lreal1:=fbMeter[1].stDataEMOutPowerDelay.lrPowerTotal;
lreal2:=fbMeter[2].stDataEMOutPowerDelay.lrPowerTotal;
lreal3:=fbMeter[3].stDataEMOutPowerDelay.lrPowerTotal;
lreal4:=fbMeter[4].stDataEMOutPowerDelay.lrPowerTotal;
lreal5:=fbMeter[5].stDataEMOutPowerDelay.lrPowerTotal;
lreal6:=fbMeter[6].stDataEMOutPowerDelay.lrPowerTotal;
lreal7:=fbMeter[7].stDataEMOutPowerDelay.lrPowerTotal;
lreal8:=fbMeter[8].stDataEMOutPowerDelay.lrPowerTotal;
lreal9:=fbMeter[9].stDataEMOutPowerDelay.lrPowerTotal;
lreal10:=fbMeter[10].stDataEMOutPowerDelay.lrPowerTotal;
lreal11:=fbMeter[11].stDataEMOutPowerDelay.lrPowerTotal;
lreal12:=fbMeter[12].stDataEMOutPowerDelay.lrPowerTotal;
lreal13:=fbMeter[13].stDataEMOutPowerDelay.lrPowerTotal;
lreal14:=fbMeter[14].stDataEMOutPowerDelay.lrPowerTotal;
lreal15:=fbMeter[15].stDataEMOutPowerDelay.lrPowerTotal;
lreal16:=fbMeter[16].stDataEMOutPowerDelay.lrPowerTotal;
lreal17:=fbMeter[17].stDataEMOutPowerDelay.lrPowerTotal;
lreal18:=fbMeter[18].stDataEMOutPowerDelay.lrPowerTotal;
lreal19:=fbMeter[19].stDataEMOutPowerDelay.lrPowerTotal;
lreal20:=fbMeter[20].stDataEMOutPowerDelay.lrPowerTotal;

(*----------------------------------------------------------Save persistent data----------------------------------------------------------------*)

// arrPD[1](lrValue:= BOOL_TO_LREAL(bEnable), bEventBasedActive=> );
// arrPD[2](lrValue:= BYTE_TO_LREAL(byAmountOfInverters), bEventBasedActive=> );
PD_String(sText:= sIPAdress, bEventBasedActive=> );

END_FUNCTION_BLOCK

// ---- FBs/Keba/FB_ECS_Keba_P30.TcPOU
FUNCTION_BLOCK FB_ECS_Keba_P30
VAR_INPUT PERSISTENT
	///{#lynus.ag#()} //Enable the Fuctionblock and his logic
	bEnable: BOOL;
	///With True its possible to invert all received power data from the electric meter
	bPowerDataInvers: BOOL;
	///Electric Fuse Line on wich the ECS is connected => 1 2 3 (If 0 then this charging station is not connected to a Electric Fuse Line)
	byElectricFuseLine: BYTE;
	///Failsafe Current when the connection between PLC and Charging station is interrupted. 0mA = CS Off, 6000mA - 32000mA
	uiFailsafeCurrent: UINT;
	///Failsafe Timeout when the connection between PLC and Charging station is interrupted. 10 - 600 sec
	uiFailsafeTimeOut: UINT := 10;
	///Number of EMS what control this Device.
	diNrOfEMS_IN: DINT;
	///Number of the electric meter for incoming power data. (Power Data for this Device)
	diNrOfEM_IN_CS: DINT;
	///IP Adress from the Keba charging station
	sIPAdress: STRING(15);
	///{#lynus.ag#()} //Setup charging station
	stSetupECS: ST_Setup_ECS;
END_VAR
VAR_OUTPUT
	///{#lynus.ag#()} //Electric charging station output data
	stDataECS: ST_ECS_Output;
	///Active Number from the Electric charging Function for using on other functions
	diNrOfECS_OUT: DINT;
	///Total Electric Power in kW read out directly from the Charging station. (Real time)
	lrTotalPowerECSRealTime: LREAL;
END_VAR
VAR
	///Function block for electric charging station
	{attribute 'hide' := ''}
	fbCS: FB_ElectricChargingStation;
	///Function block to calcualte the number of the Device
	{attribute 'hide' := ''}
	fbNumberDevice: FB_NumberOfDevice;
	///Digital Input from external loock signal
	fbDIExternalLock: FB_XL1XXX_DI;
	///Modbus Read Function (FC3)
	{attribute 'hide' := ''}
	fbMBRead_FC3: FB_MBReadRegs;
	///Modbus Write Function (FC6)
	{attribute 'hide' := ''}
	fbMBWrite_FC6: FB_MBWriteSingleReg;
	///Convert Word to Dword
	{attribute 'hide' := ''}
	fbConvertWordToDword: FB_CV_WORD_TO_DWORD;
	///Timer for Delay between Requests
	{attribute 'hide' := ''}
	timDelay: TON;
	///Timer for Timeout
	{attribute 'hide' := ''}
	timTimeout: TON;
	///Timer to dissable the Function after Lynus_Standards.Constants_General.tTimeDissableLynusFunctions Days without connection to the Lynus Cloud
	{attribute 'hide' := ''}
	timDissableFunctions: TON;
	///Timer to try reset the connection Flag on the GVL. (When somebody delete the Connection Function and make only a onlinechange)
	{attribute 'hide' := ''}
	timResetConnectionOnGVL: TON;
	///Charging Time
	{attribute 'hide' := ''}
	timChTimeSocket: TON;
	///Timer to start the state machine with Daley after enabling or after the system ist restartet
	{attribute 'hide' := ''}
	timDelayStart: TON;
	///Timer to Close the Socket after to much Errors
	{attribute 'hide' := ''}
	timCloseSocket: TON;
	///Internal positive Edge
	{attribute 'hide' := ''}
	FPError_FC_3: R_TRIG;
	///Internal positive Edge
	{attribute 'hide' := ''}
	FPError_FC_6: R_TRIG;
	///Internal positive Edge
	{attribute 'hide' := ''}
	FPEnable: R_TRIG;
	///Function to save persistent data
	{attribute 'hide' := ''}
	arrPD: ARRAY[1..16] OF FB_PersistentData_Number;
	///Function to save persistent string data
	{attribute 'hide' := ''}
	fbPDString: FB_PersistentData_String;
	///Buffer with Data from FC3
	{attribute 'hide' := ''}
	arrBuffer_FC3: ARRAY[1..2] OF WORD;
	///Error State from the charging station
	{attribute 'hide' := ''}
	bErrorCS: BOOL;
	///Modbus TCP Function Error Counter																	
	{attribute 'hide' := ''}
	byMBTCPErrorCounter: BYTE;
	///Wait in Step before start to clean data on PLC
	{attribute 'hide' := ''}
	byWaitInStep: BYTE;
	///State machine to handle the data on the GVL
	{attribute 'hide' := ''}
	iStateGVLData: INT;
	///State machine for read out Data over Modbus TCP
	{attribute 'hide' := ''}
	iStateModbusRead: INT;
	///State machine for write Data over Modbus TCP
	{attribute 'hide' := ''}
	iStateModbusWrite: INT;
	///State machine for error out Data over Modbus TCP	
	{attribute 'hide' := ''}
	iStateModbusError: INT;
	///Variable to compare the state machine variable to set or reset the timeout timer
	{attribute 'hide' := ''}
	iStateModbus_CP: INT;
	///Number of active batterys
	{attribute 'hide' := ''}
	diNumberOfActiveBatterys: DINT;
	///Number of battery inverters that work in Emergency Power operation 
	{attribute 'hide' := ''}
	diNumberOfBatteryInverterInEPO: DINT;
	///Loop to clean old data on GVL
	{attribute 'hide' := ''}
	diLPForGVL: DINT;
	///Counter to clean old data on GVL
	{attribute 'hide' := ''}
	diCounterForGVL: DINT;
	///Sum of the SOC from all batterys
	{attribute 'hide' := ''}
	dwSumSOC: DWORD;
	///Charging State from the Keba Charger
	{attribute 'hide' := ''}
	dwChargingState: DWORD;
	///Cable State from the Keba Charger
	{attribute 'hide' := ''}
	dwCableState: DWORD;
	///Error Code from the Keba Charger
	{attribute 'hide' := ''}
	dwErrorCode: DWORD;
	///Power from the ECS in W 
	{attribute 'hide' := ''}
	rPowerECS: REAL;
	///Energy Counter Consumption in Wh
	{attribute 'hide' := ''}
	lrTotalCounterEnergy_Consumption: LREAL;
	///Charged Energy from the active Session in Wh
	{attribute 'hide' := ''}
	lrChargedEnergySession: LREAL;
	///Loop to check some data from batterys
	{attribute 'hide' := ''}
	liLPBatteryData: LINT;
	///Loop to check if 1 or more battery inverters build a island grid
	{attribute 'hide' := ''}
	liLPInEPO: LINT;
END_VAR
VAR PERSISTENT
	///Number of EMS what control this Device to compare with the original
	{attribute 'conditionalshow' := ''}
	diNrOfEMS_IN_CP: DINT;
END_VAR

//Creator : Kai Ebensperger
//Company : Lynus AG
//Date : 15.07.2022
//Version : 1.0.0.0

//With this Funcition its possible to communicate with a Keba P30 Charging station over Modbus TCP.
//Support the C-Series from Version 3.10.16 or higher
//Support the X-Series from Version 1.11 or higher
//Its possible to controll the charging station over the charge current
//When the Function send 0 Ampere is switched of, then the charging station is blocked and its not possible to charge
//The Communication is not so fast because in the Documentation they write that we can read every 500MS but we can write onle ever 5 seconds.
//We can read only 1 Register at each command. Its not possible to read more Registers with 1 command
//The Unit ID is always 255
//Also the Settings for Fail Save is includes in ths Fuction. The Failsave Current is set to uiFailsafeCurrent.
//Failsafe takes effect when the connection between the PLC and the charging station is interrupted. Timout is uiFailsafeTimeOut in seconds.

//Versions that are supported : 1.3

//NOTE for diNr.....Designation => 
//_IN = Here Data come in from other Functions or go out to other functions about the GVL
//_OUT = Here Data go out to other functions about the GVL

(*--------------------------------------------------------------------------------------------Limits-------------------------------------------------------------------------------------*)

diNrOfEMS_IN := LIMIT(0,diNrOfEMS_IN,Constants_Energy.diMaxNumberOfEMS);
	diNrOfEM_IN_CS := LIMIT(0,diNrOfEM_IN_CS,Constants_Energy.diMaxNumberOfElectricMeters);
		byElectricFuseLine := LIMIT(0,byElectricFuseLine,30);
			IF uiFailsafeCurrent > 0 THEN 
				uiFailsafeCurrent := LIMIT(6000,uiFailsafeCurrent,32000);
			END_IF 
				uiFailsafeTimeOut := LIMIT(10,uiFailsafeTimeOut,600);	
		
(*------------------------------------------------------------------Power Data----------------------------------------------------------------------------*)

IF diNrOfEM_IN_CS <> 0 THEN
	//Energy Session Input data
	fbCS.bCalculateEnergySession := FALSE;
	fbCS.arrSocketPowerECS[1] := 0;
	fbCS.arrSocketPowerECS[2] := 0;
	fbCS.arrSocketPowerECS[3] := 0;
	fbCS.arrSocketPowerECS[4] := 0;
	fbCS.arrSocketEnergySession[1] := 0;
	fbCS.arrSocketEnergySession[2] := 0;
	fbCS.arrSocketEnergySession[3] := 0;
	fbCS.arrSocketEnergySession[4] := 0;
		IF NOT bPowerDataInvers THEN
			//Energy meter input data for cs Function block
			fbCS.lrCounterEnergyT1_Consumption := Lynus_Standards.GVL_Energy.stDataElectricMeters[diNrOfEM_IN_CS].lrCounterEnergyT1_Production * 1000;
			fbCS.lrCounterEnergyT2_Consumption := Lynus_Standards.GVL_Energy.stDataElectricMeters[diNrOfEM_IN_CS].lrCounterEnergyT2_Production * 1000;
			fbCS.lrCounterEnergyT1_Production := Lynus_Standards.GVL_Energy.stDataElectricMeters[diNrOfEM_IN_CS].lrCounterEnergyT1_Consumption * 1000;
			fbCS.lrCounterEnergyT2_Production := Lynus_Standards.GVL_Energy.stDataElectricMeters[diNrOfEM_IN_CS].lrCounterEnergyT1_Consumption * 1000;
			fbCS.lrTotalCounterEnergy_Consumption := Lynus_Standards.GVL_Energy.stDataElectricMeters[diNrOfEM_IN_CS].lrTotalCounterEnergy_Production * 1000;
			fbCS.lrTotalCounterEnergy_Production := Lynus_Standards.GVL_Energy.stDataElectricMeters[diNrOfEM_IN_CS].lrTotalCounterEnergy_Consumption * 1000;
				fbCS.lrTotalPowerECS := (Lynus_Standards.GVL_Energy.stDataElectricMeters[diNrOfEM_IN_CS].lrPower * 1000) * - 1;
			ELSE
			//Energy meter input data for cs Function block
			fbCS.lrCounterEnergyT1_Consumption := Lynus_Standards.GVL_Energy.stDataElectricMeters[diNrOfEM_IN_CS].lrCounterEnergyT1_Consumption * 1000;
			fbCS.lrCounterEnergyT2_Consumption := Lynus_Standards.GVL_Energy.stDataElectricMeters[diNrOfEM_IN_CS].lrCounterEnergyT2_Consumption * 1000;
			fbCS.lrCounterEnergyT1_Production := Lynus_Standards.GVL_Energy.stDataElectricMeters[diNrOfEM_IN_CS].lrCounterEnergyT1_Production * 1000;
			fbCS.lrCounterEnergyT2_Production := Lynus_Standards.GVL_Energy.stDataElectricMeters[diNrOfEM_IN_CS].lrCounterEnergyT2_Production * 1000;
			fbCS.lrTotalCounterEnergy_Consumption := Lynus_Standards.GVL_Energy.stDataElectricMeters[diNrOfEM_IN_CS].lrTotalCounterEnergy_Consumption * 1000;
			fbCS.lrTotalCounterEnergy_Production := Lynus_Standards.GVL_Energy.stDataElectricMeters[diNrOfEM_IN_CS].lrTotalCounterEnergy_Production * 1000;
				fbCS.lrTotalPowerECS := Lynus_Standards.GVL_Energy.stDataElectricMeters[diNrOfEM_IN_CS].lrPower * 1000;
		END_IF
ELSE
	//Energy meter input data for cs Function block
	fbCS.lrCounterEnergyT1_Consumption := lrTotalCounterEnergy_Consumption;
	fbCS.lrCounterEnergyT2_Consumption := 0;
	fbCS.lrCounterEnergyT1_Production := 0;
	fbCS.lrCounterEnergyT2_Production := 0;
	fbCS.lrTotalCounterEnergy_Consumption := lrTotalCounterEnergy_Consumption;
	fbCS.lrTotalCounterEnergy_Production := 0;
		fbCS.lrTotalPowerECS := rPowerECS;
	//Energy Session Input data
	fbCS.bCalculateEnergySession := FALSE;
	fbCS.arrSocketPowerECS[1] := rPowerECS;
	fbCS.arrSocketPowerECS[2] := 0;
	fbCS.arrSocketPowerECS[3] := 0;
	fbCS.arrSocketPowerECS[4] := 0;
	fbCS.arrSocketEnergySession[1] := lrChargedEnergySession;
	fbCS.arrSocketEnergySession[2] := 0;
	fbCS.arrSocketEnergySession[3] := 0;
	fbCS.arrSocketEnergySession[4] := 0;
END_IF			

(*-------------------------------------------------------------Calcualte the number of ECS---------------------------------------------------------------*)

fbNumberDevice(
	diActualNumberOfDevices:= Lynus_Standards.GVL_Energy.stNumberOfDevices.diNumberOfECS, 
	diMaxNumberOfDevices:= Constants_Energy.diMaxNumberOfElectricChargingStations, 
	udiCounterOnlineChange:= TwinCAT_SystemInfoVarList._AppInfo.OnlineChangeCnt, 
	bNumberIsCalculatet=> , 
	bFPNumberIsCalculatet=> , 
	bOnlineChange=> , 
	diNumberForThisDevice=> diNrOfECS_OUT, 
	diNumberOfTotalDevices=> );

//Write new Numer on GVL
IF fbNumberDevice.bFPNumberIsCalculatet THEN
	Lynus_Standards.GVL_Energy.stNumberOfDevices.diNumberOfECS := fbNumberDevice.diNumberOfTotalDevices;	
END_IF 

//Delete old Number on GVL
IF fbNumberDevice.bOnlineChange THEN 
	Lynus_Standards.GVL_Energy.stNumberOfDevices.diNumberOfECS := diNrOfECS_OUT;	
		iStateGVLData := 1;
END_IF

(*-------------------------------------------------------------Service from Backend is ready and check the connection to backen for dissabel/enable Function---------------------------------------------------------------*)

//Try to reset the variable for connection on the GVL. When all is normal then the Lynus Mqtt connection function set this variable to true in the next cycle
//When we have no connection to the backend then after Lynus_Standards.Constants_General.tTimeDissableLynusFunctions days the Function is dissabled with all of his functionalities
timResetConnectionOnGVL(IN:= NOT timResetConnectionOnGVL.Q, PT:= T#1H, Q=> , ET=> );
	IF timResetConnectionOnGVL.Q THEN Lynus_Standards.GVL_Communicator.bStateConnectionToEnableFunctions := FALSE; END_IF
		IF NOT Lynus_Standards.GVL_Communicator.bStateConnectionToEnableFunctions THEN timDissableFunctions.IN := TRUE; ELSE timDissableFunctions.IN := FALSE; END_IF  
			timDissableFunctions(IN:= , PT:= Lynus_Standards.Constants_General.tTimeDissableLynusFunctions, Q=> , ET=> );
			
(*--------------------------------------------------------------------------------------------State Machine Read--------------------------------------------------------------------------------------*)

//Timer for Delay
timDelay(IN:= , PT:= T#750MS, Q=> , ET=> );

//Timer for Timeout in Statemachine
IF (iStateModbusRead > 0 AND iStateModbusRead <= 7 AND iStateModbusRead = iStateModbus_CP) OR
		(iStateModbusWrite > 0 AND iStateModbusWrite <= 2 AND iStateModbusWrite = iStateModbus_CP) THEN
			timTimeout.IN := TRUE;
ELSE	
			timTimeout.IN := FALSE;
END_IF
	//Timeout Timer is dissabled when the Init Step is aktiv or the function is not enabled
	IF (iStateModbusRead = 0 AND iStateModbusWrite = 0) OR NOT bEnable THEN timTimeout.IN := FALSE; END_IF
		timTimeout(IN:= , PT:= T#10S, Q=> , ET=> );

//Enable with Delay that not all sockets have to be created at the same time
timDelayStart(IN:= bEnable, PT:= T#20MS * diNrOfECS_OUT, Q=> , ET=> );
	FPEnable(CLK:= timDelayStart.Q, Q=> );

IF FPEnable.Q AND iStateModbusRead = 0 AND iStateModbusWrite = 0 THEN iStateModbusRead := 1; END_IF		
		
//Not Enabled
IF NOT bEnable THEN iStateModbusRead := 0; iStateModbusError := 0; iStateModbusWrite := 0; END_IF		
		
CASE iStateModbusRead OF

	0://Init Step 
		iStateModbus_CP := 0;
			timDelay.IN := FALSE;
				fbMBRead_FC3.bExecute := FALSE;
					fbMBWrite_FC6.bExecute := FALSE;
						rPowerECS := 0;
							dwChargingState := 0;
								dwCableState := 0;	
									lrChargedEnergySession := 0;
	
	1://Charging State (Register 1000) !!!!Maybe 0 or 1....test it. Then change also the other Register Adresses!!!!!
		iStateModbus_CP := iStateModbusRead;

		//Start Read
		fbMBRead_FC3.nQuantity := 2;
			fbMBRead_FC3.nMBAddr := 1000;
				fbMBRead_FC3.bExecute := TRUE;
					fbMBRead_FC3.nUnitID := 255;
			
		IF fbMBRead_FC3.bBusy THEN timDelay.IN := TRUE; END_IF
		
		//Wait for Delay, copy Data and then next step
		IF NOT fbMBRead_FC3.bBusy AND NOT fbMBRead_FC3.bError AND timDelay.Q THEN
			//Charging State
			fbConvertWordToDword(wInputValue_1:= arrBuffer_FC3[1], wInputValue_2:= arrBuffer_FC3[2], eByteOrderForConvert:= eByteOrder.eBigEndian, dwOutputValue =>);
				dwChargingState := fbConvertWordToDword.dwOutputValue;
			
			//Go to Next Step
			fbMBRead_FC3.bExecute := FALSE;
				timDelay.IN := FALSE;		
					iStateModbusRead := 2;
		END_IF	

		//Error or Timeout
		IF FPError_FC_3.Q OR timTimeout.Q THEN
			iStateModbusError := 300;
		END_IF	
		
	2://Cable State (Register 1004)
		iStateModbus_CP := iStateModbusRead;

		//Start Read
		fbMBRead_FC3.nQuantity := 2;
			fbMBRead_FC3.nMBAddr := 1004;
				fbMBRead_FC3.bExecute := TRUE;
					fbMBRead_FC3.nUnitID := 255;
			
		IF fbMBRead_FC3.bBusy THEN timDelay.IN := TRUE; END_IF
		
		//Wait for Delay, copy Data and then next step
		IF NOT fbMBRead_FC3.bBusy AND NOT fbMBRead_FC3.bError AND timDelay.Q THEN
			//Cable State
			fbConvertWordToDword(wInputValue_1:= arrBuffer_FC3[1], wInputValue_2:= arrBuffer_FC3[2], eByteOrderForConvert:= eByteOrder.eBigEndian, dwOutputValue =>);
				dwCableState := fbConvertWordToDword.dwOutputValue;
			//Go to Next Step
			fbMBRead_FC3.bExecute := FALSE;
				timDelay.IN := FALSE;		
					iStateModbusRead := 3;
		END_IF	

		//Error or Timeout
		IF FPError_FC_3.Q OR timTimeout.Q THEN
			iStateModbusError := 300;
		END_IF	
		
	3://Error Code (Register 1006)
		iStateModbus_CP := iStateModbusRead;

		//Start Read
		fbMBRead_FC3.nQuantity := 2;
			fbMBRead_FC3.nMBAddr := 1006;
				fbMBRead_FC3.bExecute := TRUE;
					fbMBRead_FC3.nUnitID := 255;
			
		IF fbMBRead_FC3.bBusy THEN timDelay.IN := TRUE; END_IF
		
		//Wait for Delay, copy Data and then next step
		IF NOT fbMBRead_FC3.bBusy AND NOT fbMBRead_FC3.bError AND timDelay.Q THEN
			//Error Code
			fbConvertWordToDword(wInputValue_1:= arrBuffer_FC3[1], wInputValue_2:= arrBuffer_FC3[2], eByteOrderForConvert:= eByteOrder.eBigEndian, dwOutputValue =>);
				dwErrorCode := fbConvertWordToDword.dwOutputValue;
			//Go to Next Step
			fbMBRead_FC3.bExecute := FALSE;
				timDelay.IN := FALSE;		
					iStateModbusRead := 4;
		END_IF	

		//Error or Timeout
		IF FPError_FC_3.Q OR timTimeout.Q THEN
			iStateModbusError := 300;
		END_IF	
		
	4://Active Power (Register 1020)
		iStateModbus_CP := iStateModbusRead;

		//Start Read
		fbMBRead_FC3.nQuantity := 2;
			fbMBRead_FC3.nMBAddr := 1020;
				fbMBRead_FC3.bExecute := TRUE;
					fbMBRead_FC3.nUnitID := 255;
			
		IF fbMBRead_FC3.bBusy THEN timDelay.IN := TRUE; END_IF
		
		//Wait for Delay, copy Data and then next step
		IF NOT fbMBRead_FC3.bBusy AND NOT fbMBRead_FC3.bError AND timDelay.Q THEN
			//Active Power in mW
			fbConvertWordToDword(wInputValue_1:= arrBuffer_FC3[1], wInputValue_2:= arrBuffer_FC3[2], eByteOrderForConvert:= eByteOrder.eBigEndian, dwOutputValue =>);
				rPowerECS := DWORD_TO_REAL(fbConvertWordToDword.dwOutputValue);
					rPowerECS := rPowerECS / 1000;	
			//Go to Next Step
			fbMBRead_FC3.bExecute := FALSE;
				timDelay.IN := FALSE;		
					iStateModbusRead := 5;
		END_IF	

		//Error or Timeout
		IF FPError_FC_3.Q OR timTimeout.Q THEN
			iStateModbusError := 300;
		END_IF	
	
	5://Total Energy (Register 1036)
		iStateModbus_CP := iStateModbusRead;

		//Start Read
		fbMBRead_FC3.nQuantity := 2;
			fbMBRead_FC3.nMBAddr := 1036;
				fbMBRead_FC3.bExecute := TRUE;
					fbMBRead_FC3.nUnitID := 255;
			
		IF fbMBRead_FC3.bBusy THEN timDelay.IN := TRUE; END_IF
		
		//Wait for Delay, copy Data and then next step
		IF NOT fbMBRead_FC3.bBusy AND NOT fbMBRead_FC3.bError AND timDelay.Q THEN
			//Total Energy in Wh
			fbConvertWordToDword(wInputValue_1:= arrBuffer_FC3[1], wInputValue_2:= arrBuffer_FC3[2], eByteOrderForConvert:= eByteOrder.eBigEndian, dwOutputValue =>);
				lrTotalCounterEnergy_Consumption := DWORD_TO_LREAL(fbConvertWordToDword.dwOutputValue);
			//Go to Next Step
			fbMBRead_FC3.bExecute := FALSE;
				timDelay.IN := FALSE;		
					iStateModbusRead := 6;
		END_IF	

		//Error or Timeout
		IF FPError_FC_3.Q OR timTimeout.Q THEN
			iStateModbusError := 300;
		END_IF	
		
	6://Charged Energy from current charging session (Register 1502)
		iStateModbus_CP := iStateModbusRead;

		//Start Read
		fbMBRead_FC3.nQuantity := 2;
			fbMBRead_FC3.nMBAddr := 1502;
				fbMBRead_FC3.bExecute := TRUE;
					fbMBRead_FC3.nUnitID := 255;
			
		IF fbMBRead_FC3.bBusy THEN timDelay.IN := TRUE; END_IF
		
		//Wait for Delay, copy Data and then next step
		IF NOT fbMBRead_FC3.bBusy AND NOT fbMBRead_FC3.bError AND timDelay.Q THEN
			//Total Energy in Wh
			fbConvertWordToDword(wInputValue_1:= arrBuffer_FC3[1], wInputValue_2:= arrBuffer_FC3[2], eByteOrderForConvert:= eByteOrder.eBigEndian, dwOutputValue =>);
				lrChargedEnergySession := DWORD_TO_LREAL(fbConvertWordToDword.dwOutputValue);
			//Go to Next Step
			fbMBRead_FC3.bExecute := FALSE;
				timDelay.IN := FALSE;		
					iStateModbusRead := 7;
		END_IF	

		//Error or Timeout
		IF FPError_FC_3.Q OR timTimeout.Q THEN
			iStateModbusError := 300;
		END_IF	
		
	7://Wait 1 Step to reset the delay counter befor start to write
		iStateModbus_CP := iStateModbusRead;
		
			iStateModbusWrite := 1;
				//-1 because 0 is the Init Step for Read
				iStateModbusRead := - 1;
				
			//Error on Master, changes on Inputs or Timeout
		 	IF timTimeout.Q THEN 
				iStateModbusError := 300;	 
			END_IF
	
END_CASE

(*------------------------------------------------------------------Error and Warning----------------------------------------------------------------------------*)	
 
IF dwChargingState = 4 OR dwErrorCode <> 0 THEN bErrorCS := TRUE; ELSE bErrorCS := FALSE; END_IF

IF timDissableFunctions.Q THEN fbCS.bWarning := TRUE; fbCS.iWarningCode := 0; ELSE fbCS.bWarning := FALSE; END_IF   
	IF Lynus_Standards.GVL_Energy.stNumberOfDevices.diNumberOfECS > Constants_Energy.diMaxNumberOfElectricChargingStations OR bErrorCS OR byMBTCPErrorCounter > 10 THEN 
		fbCS.bError := TRUE;
	ELSE 
		fbCS.bError := FALSE;
			fbCS.iErrorCode := 0;
	END_IF

IF Lynus_Standards.GVL_Energy.stNumberOfDevices.diNumberOfECS > Constants_Energy.diMaxNumberOfElectricChargingStations THEN fbCS.iErrorCode := 1;
ELSIF bErrorCS OR byMBTCPErrorCounter > 10 THEN fbCS.iErrorCode := 0; END_IF

(*------------------------------------------------------------------Logic----------------------------------------------------------------------------*)

//Calcualte the total SOC if we have more then 1 battery in our system
diNumberOfActiveBatterys := 0;
	dwSumSOC := 0;
		FOR liLPBatteryData := 1 TO Constants_Energy.diMaxNumberOfBatterys BY 1 DO
			IF Lynus_Standards.GVL_Energy.stDataOfBatterys[diNrOfEMS_IN,liLPBatteryData].bEnabled THEN diNumberOfActiveBatterys := diNumberOfActiveBatterys + 1; END_IF
				dwSumSOC := dwSumSOC + Lynus_Standards.GVL_Energy.stDataOfBatterys[diNrOfEMS_IN,liLPBatteryData].dwSOC;
		END_FOR
	
IF diNumberOfActiveBatterys > 0 THEN
	fbCS.dwBatterySOC := DINT_TO_DWORD(DWORD_TO_DINT(dwSumSOC) / diNumberOfActiveBatterys);
ELSE
	fbCS.dwBatterySOC := 100;	//When we have no battery in the ems system
END_IF

//Check if one or more Batterysystems or batteryinverter make island mode
diNumberOfBatteryInverterInEPO := 0;
	FOR liLPInEPO := 1 TO Constants_Energy.diMaxNumberOfBatteryInverters BY 1 DO
		IF Lynus_Standards.GVL_Energy.stDataOfBatteryInverters[diNrOfEMS_IN,liLPInEPO].bWorkOnIslandMode THEN fbCS.bEPOIsActive := TRUE; diNumberOfBatteryInverterInEPO := diNumberOfBatteryInverterInEPO + 1; END_IF
	END_FOR 
		IF diNumberOfBatteryInverterInEPO <= 0 THEN fbCS.bEPOIsActive := FALSE; END_IF

//Digital input for external lock signal
fbDIExternalLock(bInvers:= FALSE, bSignal=> );

//Car connected to the ECS
IF dwCableState = 5 OR dwCableState = 7 THEN fbCS.bCarConnected := TRUE; ELSE fbCS.bCarConnected := FALSE; END_IF

//Charging time
IF dwChargingState = 3 OR dwCableState = 7 THEN timChTimeSocket.IN := TRUE; ELSE timChTimeSocket.IN := FALSE; END_IF

IF timChTimeSocket.IN THEN fbCS.arrSocketChargingTimeInput[1] := TIME_TO_REAL(timChTimeSocket.ET) / 60000; END_IF
fbCS.arrSocketChargingTimeInput[2] := 0;
fbCS.arrSocketChargingTimeInput[3] := 0;
fbCS.arrSocketChargingTimeInput[4] := 0;

timChTimeSocket(IN:= , PT:= T#24H, Q=> , ET=> );

//Mode 3 State
//Default set to No Informantion
fbCS.arrSocketMode3StateECS[1] := '';
	//Ready or Free
	IF dwChargingState = 2 THEN fbCS.arrSocketMode3StateECS[1] := 'A'; END_IF
	//Car Connected
	IF dwCableState = 5 OR dwCableState = 7 THEN fbCS.arrSocketMode3StateECS[1] := 'B1'; END_IF
	//Charging
	IF dwChargingState = 3 OR dwCableState = 7 THEN fbCS.arrSocketMode3StateECS[1] := 'C2'; END_IF
	//Error
	IF dwChargingState = 4 OR dwErrorCode <> 0 THEN fbCS.arrSocketMode3StateECS[1] := 'F'; END_IF 

fbCS.arrSocketMode3StateECS[2] := '';
fbCS.arrSocketMode3StateECS[3] := '';
fbCS.arrSocketMode3StateECS[4] := '';

//SOC Car
fbCS.arrSOCCar[1] := 0;
fbCS.arrSOCCar[2] := 0;
fbCS.arrSOCCar[3] := 0;
fbCS.arrSOCCar[4] := 0;

//Functionblock ECS
fbCS(
	bEnable:= bEnable AND NOT timDissableFunctions.Q, 
	bError:= ,
	bWarning := ,
	bEPOIsActive:= , 
	bExternalLock:= fbDIExternalLock.bSignal, 
	bCarConnected:= , 
	bWriteWithDelay:= TRUE, 
	bCalculateEnergySession:= ,
	iErrorCode:= , 
	iWarningCode:= , 
	arrSocketChargingTimeInput:= ,
	arrSOCCar:= , 
	dwBatterySOC:= , 
	lrTotalCounterEnergy_Consumption:= , 
	lrTotalCounterEnergy_Production:= , 
	lrCounterEnergyT1_Consumption:= , 
	lrCounterEnergyT2_Consumption:= , 
	lrCounterEnergyT1_Production:= , 
	lrCounterEnergyT2_Production:= , 
	lrTotalPowerECS:= , 
	arrSocketEnergySession:= ,
	rTargetPower:= Lynus_Standards.GVL_Energy.stDataElectricChargingStations[diNrOfEMS_IN,diNrOfECS_OUT].rTargetPowerEMS, 
	rSupplyVoltage:= 692, 
	rMinCurrent:= 6, 
	tTimDelayOutput:= T#5S, 
	tDelayError:= T#5S,
	arrSocketMode3StateECS:= ,
	arrSocketPowerECS:= ,
	stSetupECS:= stSetupECS, 
	stDataECSOut=> , 
	stDataECSOutDelay=> stDataECS);

//Real time Power for Output
lrTotalPowerECSRealTime := fbCS.stDataECSOut.lrTotalPower;
	
(*------------------------------------------------------------------------------------------State Machine Write---------------------------------------------------------------------------------------------*)	

CASE iStateModbusWrite OF	

	1://Set the charging current (Reg 5004)
		iStateModbus_CP := iStateModbusWrite;
		
			fbMBWrite_FC6.nMBAddr := 5004;
				fbMBWrite_FC6.bExecute := TRUE;
					fbMBWrite_FC6.nUnitID := 255;
						//Charge Current in mA
						fbMBWrite_FC6.nValue := REAL_TO_WORD(fbCS.stDataECSOut.rTargetChargeCurrent * 1000);
		
		IF fbMBWrite_FC6.bBusy THEN timDelay.IN := TRUE; END_IF

		//Wait for Delay and then next step
		IF NOT fbMBWrite_FC6.bBusy AND NOT fbMBWrite_FC6.bError AND timDelay.Q THEN
			fbMBWrite_FC6.bExecute := FALSE;
				timDelay.IN := FALSE;
					//Go to Next Step
					iStateModbusWrite := 2;
		END_IF
				
		//Error or Timout
		IF FPError_FC_6.Q OR timTimeout.Q THEN
			iStateModbusError := 300;
		END_IF
	
	2://Enable/Dissable Charging station (Reg 5014)
		iStateModbus_CP := iStateModbusWrite;
		
			fbMBWrite_FC6.nMBAddr := 5014;
				fbMBWrite_FC6.bExecute := TRUE;
					fbMBWrite_FC6.nUnitID := 255;
						//Enable and Dissable the Charging station
						IF fbCS.stDataECSOut.rTargetChargeCurrent <> 0 THEN 
							//Enable
							fbMBWrite_FC6.nValue := 1;
						ELSE
							//Dissable
							fbMBWrite_FC6.nValue := 0;
						END_IF
		
		IF fbMBWrite_FC6.bBusy THEN timDelay.IN := TRUE; END_IF

		//Wait for Delay and then next step
		IF NOT fbMBWrite_FC6.bBusy AND NOT fbMBWrite_FC6.bError AND timDelay.Q THEN
			fbMBWrite_FC6.bExecute := FALSE;
				timDelay.IN := FALSE;
					//Go to Next Step
					iStateModbusWrite := 3;
		END_IF
				
		//Error or Timout
		IF FPError_FC_6.Q OR timTimeout.Q THEN
			iStateModbusError := 300;
		END_IF
		
	3://Failsafe current (Reg 5016)
		iStateModbus_CP := iStateModbusWrite;
		
			fbMBWrite_FC6.nMBAddr := 5016;
				fbMBWrite_FC6.bExecute := TRUE;
					fbMBWrite_FC6.nUnitID := 255;
						//Failsafe current in mA
						fbMBWrite_FC6.nValue := uiFailsafeCurrent;
	
		IF fbMBWrite_FC6.bBusy THEN timDelay.IN := TRUE; END_IF

		//Wait for Delay and then next step
		IF NOT fbMBWrite_FC6.bBusy AND NOT fbMBWrite_FC6.bError AND timDelay.Q THEN
			fbMBWrite_FC6.bExecute := FALSE;
				timDelay.IN := FALSE;
					//Go to Next Step
					iStateModbusWrite := 3;
		END_IF
				
		//Error or Timout
		IF FPError_FC_6.Q OR timTimeout.Q THEN
			iStateModbusError := 300;
		END_IF	
		
	4://Failsafe Timeout (Reg 5018)
		iStateModbus_CP := iStateModbusWrite;
		
			fbMBWrite_FC6.nMBAddr := 5018;
				fbMBWrite_FC6.bExecute := TRUE;
					fbMBWrite_FC6.nUnitID := 255;
						//Failsafe Timeout in sec.
						fbMBWrite_FC6.nValue := uiFailsafeTimeOut;
	
		IF fbMBWrite_FC6.bBusy THEN timDelay.IN := TRUE; END_IF

		//Wait for Delay and then next step
		IF NOT fbMBWrite_FC6.bBusy AND NOT fbMBWrite_FC6.bError AND timDelay.Q THEN
			fbMBWrite_FC6.bExecute := FALSE;
				timDelay.IN := FALSE;
					byMBTCPErrorCounter := 0; 
						//Restart from new with the Read out part
						iStateModbusRead := 1;
							iStateModbusWrite := 0;
		END_IF
				
		//Error or Timout
		IF FPError_FC_6.Q OR timTimeout.Q THEN
			iStateModbusError := 300;
		END_IF	
		
END_CASE	
	
(*------------------------------------------------------------------------------------------State Machine Error---------------------------------------------------------------------------------------------*)	

CASE iStateModbusError OF
	
	300://Error
		iStateModbus_CP := iStateModbusError;
			timDelay.IN := FALSE;
				fbMBRead_FC3.bExecute := FALSE;
					fbMBWrite_FC6.bExecute := FALSE;
						byMBTCPErrorCounter := byMBTCPErrorCounter + 1;
							byMBTCPErrorCounter := LIMIT(0,byMBTCPErrorCounter,11); 		
								//Restart from new with the Read out part after an Error
								IF byMBTCPErrorCounter < 10 THEN
									iStateModbusRead := 1;	
										iStateModbusError := 0;
											iStateModbusWrite := 0;
								ELSE
									//Wait here in the Error State for the Delay Timer and then we dont have a Timeout Error
									iStateModbusRead := - 1;
										iStateModbusWrite := - 1;
											//Start from New when the Delay is paste
											IF timCloseSocket.Q THEN
												iStateModbusRead := 1;	
													iStateModbusError := 0;
														iStateModbusWrite := 0;	
															byMBTCPErrorCounter := 0;
											END_IF
								END_IF
						
END_CASE

//Timer to close the Socket after to much TCP Errors and reopen a new one
timCloseSocket(IN:= byMBTCPErrorCounter > 10 AND fbCS.stDataECSOut.bEnabled, PT:= T#1M, Q=> , ET=> );

(*------------------------------------------------------------------------------------------Modbus TCP Functions---------------------------------------------------------------------------------------------*)

fbMBRead_FC3(sIPAddr:= sIPAdress, nTCPPort:= 502,cbLength:= SIZEOF(arrBuffer_FC3), pDestAddr:= ADR(arrBuffer_FC3), tTimeout:= T#5S );
	FPError_FC_3(CLK:= fbMBRead_FC3.bError, Q=> );		

fbMBWrite_FC6(sIPAddr:= sIPAdress, nTCPPort:= 502, tTimeout:= T#5S);	
	FPError_FC_6(CLK:= fbMBWrite_FC6.bError, Q=> );

(*-----------------------------------------------------------Handle data to Global structure for electric charging stations-----------------------------------------------------------------*)

//Delte al old Data on GVL after a online change or change on the variable diNrOfEMS_IDOD
IF diNrOfEMS_IN <> diNrOfEMS_IN_CP AND iStateGVLData = 0 THEN iStateGVLData := 10; END_IF 

CASE iStateGVLData OF
	
	0://Init Step
		byWaitInStep := 0;
			diCounterForGVL := 1;
	
	1://Wait for 4 Steps before clean al Data on GVL
		byWaitInStep := byWaitInStep + 1;
			IF byWaitInStep >= 4 AND fbNumberDevice.bNumberIsCalculatet THEN iStateGVLData := 2; END_IF
				//To much Devices, back to the Init step
				IF byWaitInStep >= 4 AND NOT fbNumberDevice.bNumberIsCalculatet THEN iStateGVLData := 0; END_IF	
			
	2://Clear all Data in GVL
		FOR diLPForGVL := 1 TO Constants_Energy.diMaxNumberOfEMS BY 1 DO 
			Lynus_Standards.GVL_Energy.stDataElectricChargingStations[diLPForGVL,diCounterForGVL].bEnabled := FALSE;
				Lynus_Standards.GVL_Energy.stDataElectricChargingStations[diLPForGVL,diCounterForGVL].bIsControllable := FALSE;
					Lynus_Standards.GVL_Energy.stDataElectricChargingStations[diLPForGVL,diCounterForGVL].byErrorWarning := 0;
						Lynus_Standards.GVL_Energy.stDataElectricChargingStations[diLPForGVL,diCounterForGVL].byPriority := 0;
							Lynus_Standards.GVL_Energy.stDataElectricChargingStations[diLPForGVL,diCounterForGVL].lrPower := 0;
								Lynus_Standards.GVL_Energy.stDataElectricChargingStations[diLPForGVL,diCounterForGVL].lrPowerConsumption := 0;
									Lynus_Standards.GVL_Energy.stDataElectricChargingStations[diLPForGVL,diCounterForGVL].lrPowerProduction := 0;
										Lynus_Standards.GVL_Energy.stDataElectricChargingStations[diLPForGVL,diCounterForGVL].rMaxPower := 0;
											Lynus_Standards.GVL_Energy.stDataElectricChargingStations[diLPForGVL,diCounterForGVL].byElectricFuseLine := 0;
												//Set also the target value from ems back here to 0 and not in EMS function because EMS is in Standy when we have a online change (Problem when we delete a ems function and make a online change)
												Lynus_Standards.GVL_Energy.stDataElectricChargingStations[diLPForGVL,diCounterForGVL].rTargetPowerEMS := 0;	
		END_FOR
		
			//Counter for ECS
			diCounterForGVL := diCounterForGVL + 1;
				diCounterForGVL := LIMIT(0,diCounterForGVL,Constants_Energy.diMaxNumberOfElectricChargingStations);
					//Back to the init step
					IF diCounterForGVL >= Constants_Energy.diMaxNumberOfElectricChargingStations THEN iStateGVLData := 0; END_IF

	10://Clear old Data on GVL 		
		Lynus_Standards.GVL_Energy.stDataElectricChargingStations[diNrOfEMS_IN_CP,diNrOfECS_OUT].bEnabled := FALSE;
			Lynus_Standards.GVL_Energy.stDataElectricChargingStations[diNrOfEMS_IN_CP,diNrOfECS_OUT].bIsControllable := FALSE;
				Lynus_Standards.GVL_Energy.stDataElectricChargingStations[diNrOfEMS_IN_CP,diNrOfECS_OUT].byErrorWarning := 0;
					Lynus_Standards.GVL_Energy.stDataElectricChargingStations[diNrOfEMS_IN_CP,diNrOfECS_OUT].byPriority := 0;
						Lynus_Standards.GVL_Energy.stDataElectricChargingStations[diNrOfEMS_IN_CP,diNrOfECS_OUT].lrPower := 0;
							Lynus_Standards.GVL_Energy.stDataElectricChargingStations[diNrOfEMS_IN_CP,diNrOfECS_OUT].lrPowerConsumption := 0;
								Lynus_Standards.GVL_Energy.stDataElectricChargingStations[diNrOfEMS_IN_CP,diNrOfECS_OUT].lrPowerProduction := 0;
									Lynus_Standards.GVL_Energy.stDataElectricChargingStations[diNrOfEMS_IN_CP,diNrOfECS_OUT].rMaxPower := 0;
										Lynus_Standards.GVL_Energy.stDataElectricChargingStations[diNrOfEMS_IN_CP,diNrOfECS_OUT].byElectricFuseLine := 0;
									
		diNrOfEMS_IN_CP := diNrOfEMS_IN;
			//Back to the init step
			iStateGVLData := 0;

END_CASE 	 

IF diNrOfECS_OUT > 0 AND fbNumberDevice.bNumberIsCalculatet AND diNrOfEMS_IN > 0 THEN
	Lynus_Standards.GVL_Energy.stDataElectricChargingStations[diNrOfEMS_IN,diNrOfECS_OUT].bEnabled := fbCS.stDataECSOut.bEnabled;
		Lynus_Standards.GVL_Energy.stDataElectricChargingStations[diNrOfEMS_IN,diNrOfECS_OUT].bIsControllable := TRUE;
			Lynus_Standards.GVL_Energy.stDataElectricChargingStations[diNrOfEMS_IN,diNrOfECS_OUT].byErrorWarning := fbCS.stDataECSOut.byErrorWarning;
				Lynus_Standards.GVL_Energy.stDataElectricChargingStations[diNrOfEMS_IN,diNrOfECS_OUT].byPriority := fbCS.stDataECSOut.byPriority;
					Lynus_Standards.GVL_Energy.stDataElectricChargingStations[diNrOfEMS_IN,diNrOfECS_OUT].lrPower := fbCS.stDataECSOut.lrTotalPower;
						Lynus_Standards.GVL_Energy.stDataElectricChargingStations[diNrOfEMS_IN,diNrOfECS_OUT].lrPowerConsumption := fbCS.stDataECSOut.lrTotalPowerConsumption;
							Lynus_Standards.GVL_Energy.stDataElectricChargingStations[diNrOfEMS_IN,diNrOfECS_OUT].lrPowerProduction := fbCS.stDataECSOut.lrTotalPowerProduction;
								Lynus_Standards.GVL_Energy.stDataElectricChargingStations[diNrOfEMS_IN,diNrOfECS_OUT].rMaxPower := fbCS.stDataECSOut.rMaxPower;	
									Lynus_Standards.GVL_Energy.stDataElectricChargingStations[diNrOfEMS_IN,diNrOfECS_OUT].byElectricFuseLine := byElectricFuseLine;
END_IF 

(*----------------------------------------------------------Save persistent data----------------------------------------------------------------*)

arrPD[1](lrValue:= BOOL_TO_LREAL(bEnable), bEventBasedActive=> );
arrPD[2](lrValue:= BOOL_TO_LREAL(bPowerDataInvers), bEventBasedActive=> );
arrPD[3](lrValue:= DINT_TO_LREAL(diNrOfEMS_IN), bEventBasedActive=> );
arrPD[4](lrValue:= DINT_TO_LREAL(diNrOfEM_IN_CS), bEventBasedActive=> );
arrPD[5](lrValue:= BOOL_TO_LREAL(stSetupECS.bManualyOn), bEventBasedActive=> );
arrPD[6](lrValue:= BOOL_TO_LREAL(stSetupECS.bOnEmergPowerOff), bEventBasedActive=> );
arrPD[7](lrValue:= BYTE_TO_LREAL(stSetupECS.byCSMinPower), bEventBasedActive=> );
arrPD[8](lrValue:= BYTE_TO_LREAL(stSetupECS.byDisableSOC), bEventBasedActive=> );
arrPD[9](lrValue:= BYTE_TO_LREAL(stSetupECS.byEnableSOC), bEventBasedActive=> );
arrPD[10](lrValue:= BYTE_TO_LREAL(stSetupECS.byManualyTargetPower), bEventBasedActive=> );
arrPD[11](lrValue:= BYTE_TO_LREAL(stSetupECS.byPriority), bEventBasedActive=> );
arrPD[12](lrValue:= REAL_TO_LREAL(stSetupECS.rMaxPower), bEventBasedActive=> );
arrPD[13](lrValue:= DINT_TO_LREAL(diNrOfEMS_IN_CP), bEventBasedActive=> );
arrPD[14](lrValue:= BYTE_TO_LREAL(byElectricFuseLine), bEventBasedActive=> );
arrPD[15](lrValue:= UINT_TO_LREAL(uiFailsafeCurrent), bEventBasedActive=> );
arrPD[16](lrValue:= UINT_TO_LREAL(uiFailsafeTimeOut), bEventBasedActive=> );
fbPDString(sText:= sIPAdress, bEventBasedActive=> );

END_FUNCTION_BLOCK

// ---- FBs/MeteoControl/FB_BLUE_LOG_XMXC.TcPOU
FUNCTION_BLOCK FB_BLUE_LOG_XMXC
VAR_INPUT PERSISTENT
	m_Enable					: BOOL;						//Enable the Fuctionblock and his logic
	str_IPAdress				: STRING(15);				//IP Adress of the meter
	arr_byte_ID_PV				: ARRAY [1..9] OF BYTE ;		//Slave ID  PV
	
END_VAR
VAR_OUTPUT

	str_Data_Out			: ARRAY [1..9] OF str_BlueLogDataOut;
	
END_VAR
VAR
	{attribute 'hide'}
	w_Array_Received			: ARRAY[1..100] OF WORD;	// received data
	{attribute 'hide'}
	w_Adress					: WORD;						//modbus adress
	{attribute 'hide'}
	usint_Quantity				: USINT;					//Number of Words to get polled, max 100
	{attribute 'hide'}
	fbConvertWordToDword		: FB_CV_WORD_TO_DWORD;			//Convert Word to Dword
	{attribute 'hide'}
	usintSign					: USINT;						// converstion dword to real	
	{attribute 'hide'}
	intExponent					: INT;							// converstion dword to real
	{attribute 'hide'}
	realMantisse				: REAL;							// converstion dword to real
	{attribute 'hide'}
	timer_Delay					: TON;						//Timer for Delay between Requests
	{attribute 'hide'}
	timer_DelayStart			: TON;						//Timer to start the state machine with Delay after enabling or after the system ist restartet
	{attribute 'hide'}
	timer_TimeOut				: TON;						//Timer for Timeout MB Read
	{attribute 'hide'}
	iStateModbusRead			: INT;						//State machine for read out Data over Modbus RTU
	{attribute 'hide'}
	fbMBRead_FC3				: FB_MBReadRegs  ;		//Modbus Read Function (FC3)
	{attribute 'hide'}
	ftrig_PEnable				: f_trig;					//Internal positive Edge
	{attribute 'hide'}
	iStateModbusError			: INT;						//State machine for error out Data over Modbus TCP/IP	
	{attribute 'hide'}
	FPError_FC_3				: R_TRIG;					//Internal positive Edge
	{attribute 'hide'}
	arrBuffer_FC3				: ARRAY[1..100] OF WORD;		//Buffer with Data from FC3
	{attribute 'hide'}
	timer_Connection_ok			: TON;
	{attribute 'hide'}
	int_Data_Received			: INT;
	{attribute 'hide'}
	m_MBTCPError				: BOOL;
	{attribute 'hide'}
	int_Data_Received_old		: INT;
	{attribute 'hide'}
	timer_Connection_ok_TOF	: TOF;
	{attribute 'hide'}
	m_Poll_ok: BOOL;
	{attribute 'hide'}
	timer_Wait: Ton;
	{attribute 'hide'}
	int_TimeoutError: INT;
	{attribute 'hide'}
	int_FC3Error: INT;
	{attribute 'hide'}
	i: INT;
	{attribute 'hide'}
	x: INT;
	int_Poll_Count: INT:=1;
END_VAR

(*--------------------------------------------------------------------------------------------Limits-------------------------------------------------------------------------------------*)
w_Adress := 41000;
usint_Quantity := 72; 
w_Adress := LIMIT(0,w_Adress,65000);
usint_Quantity := LIMIT(1,usint_Quantity,100);
	
(*--------------------------------------------------------------------------------------------State Machine Read--------------------------------------------------------------------------------------*)

//Timer for Delay
timer_Delay(IN:= , PT:= T#50MS, Q=> , ET=> );

//Timeout Timer is dissabled when the Init Step is aktiv or the function is not enabled
IF iStateModbusRead = 0 OR NOT m_Enable THEN 
	timer_Timeout.IN := FALSE; 
END_IF
timer_Timeout(IN:= , PT:= T#1S, Q=> , ET=> );

//Enable with Delay that not all sockets have to be created at the same time
timer_DelayStart(IN:= m_Enable, PT:= T#1S, Q=> , ET=> );
ftrig_PEnable(CLK:= timer_DelayStart.Q, Q=> );

IF ftrig_PEnable.Q AND iStateModbusRead = 0 THEN 
	iStateModbusRead := 1; 
END_IF		
		
//Not Enabled
IF NOT m_Enable THEN 
	iStateModbusRead := 0; 
	iStateModbusError := 0; 
END_IF		
		
CASE iStateModbusRead OF

	0://Init Step 
		timer_Delay.IN := FALSE;
		fbMBRead_FC3.bExecute := FALSE;
		m_Poll_ok:=FALSE;
		int_Data_Received:=0;
		iStateModbusRead := 1;
		int_Poll_Count :=1;

	1: // clean the array
		FOR i:=1 TO 100 BY 1 DO
			w_Array_Received[i] := 0;
		END_FOR
		iStateModbusRead := 2;
		
	2://read the required registers
		//Start Read
		fbMBRead_FC3.nQuantity := usint_Quantity;
		fbMBRead_FC3.nMBAddr := w_Adress;
		fbMBRead_FC3.bExecute := TRUE;
		
		// Poll count 1 to 9 if next poll is not empty
		IF int_Poll_Count >= 9 THEN 
			int_Poll_Count :=1;
		ELSIF arr_byte_ID_PV[int_Poll_Count+1] >0 AND arr_byte_ID_PV[int_Poll_Count+1] <255 THEN
			int_Poll_Count := int_Poll_Count+1; 
		ELSIF arr_byte_ID_PV[int_Poll_Count+1] <=0 OR arr_byte_ID_PV[int_Poll_Count+1] >=255 THEN
			int_Poll_Count := 1; 
		END_IF
		
		
		fbMBRead_FC3.nUnitID := arr_byte_ID_PV[int_Poll_Count];
		timer_Timeout.IN := TRUE;
		IF fbMBRead_FC3.bBusy THEN 
			timer_Delay.IN := TRUE; 
		END_IF
		
		//Wait for Delay, copy Data and then next step
		IF NOT fbMBRead_FC3.bBusy AND NOT fbMBRead_FC3.bError AND timer_Delay.Q THEN
			m_Poll_ok:=TRUE;
			int_Data_Received:=int_Data_Received+1;
			m_MBTCPError := FALSE; 
			
			w_Array_Received := arrBuffer_FC3;
						
			//Go to Next Step
			timer_Timeout.IN := FALSE;
			fbMBRead_FC3.bExecute := FALSE;
			timer_Delay.IN := FALSE;		
			iStateModbusRead := 3;
		END_IF	

		//Error or Timeout
		IF FPError_FC_3.Q THEN 
			iStateModbusError := 300;
			int_FC3Error := int_FC3Error+1;
		ELSIF timer_Timeout.Q THEN  
			timer_Timeout.IN := FALSE; 	
			iStateModbusError := 300;
			int_TimeoutError := int_TimeoutError+1;
		END_IF
		
	3: // convert data
		x:=1;
			fbConvertWordToDword(wInputValue_1:= arrBuffer_FC3[x], wInputValue_2:= arrBuffer_FC3[x+1], eByteOrderForConvert:= eByteOrder.eLittleEndian , dwOutputValue=> );
			(* Sign *)
			usintSign:=BOOL_TO_USINT(fbConvertWordToDword.dwOutputValue.31);
			(* Exponent *)
			intExponent:=DWORD_TO_INT(SHR(fbConvertWordToDword.dwOutputValue,23) AND 16#FF);
			(* Mantisse *)
			realMantisse:=DWORD_TO_REAL(fbConvertWordToDword.dwOutputValue AND 16#7FFFFF);
			(* Result *)
		str_Data_Out[int_Poll_Count].real_RealPower_W := LREAL_TO_REAL((EXPT((-1),usintSign) * (1+realMantisse/8388608) * EXPT(2,intExponent-127)));
		x:=x+2;
			fbConvertWordToDword(wInputValue_1:= arrBuffer_FC3[x], wInputValue_2:= arrBuffer_FC3[x+1], eByteOrderForConvert:= eByteOrder.eLittleEndian , dwOutputValue=> );
			(* Sign *)
			usintSign:=BOOL_TO_USINT(fbConvertWordToDword.dwOutputValue.31);
			(* Exponent *)
			intExponent:=DWORD_TO_INT(SHR(fbConvertWordToDword.dwOutputValue,23) AND 16#FF);
			(* Mantisse *)
			realMantisse:=DWORD_TO_REAL(fbConvertWordToDword.dwOutputValue AND 16#7FFFFF);
			(* Result *)
		str_Data_Out[int_Poll_Count].real_ReactivePower_VAr := LREAL_TO_REAL((EXPT((-1),usintSign) * (1+realMantisse/8388608) * EXPT(2,intExponent-127)));
		x:=x+2;
			fbConvertWordToDword(wInputValue_1:= arrBuffer_FC3[x], wInputValue_2:= arrBuffer_FC3[x+1], eByteOrderForConvert:= eByteOrder.eLittleEndian , dwOutputValue=> );
			(* Sign *)
			usintSign:=BOOL_TO_USINT(fbConvertWordToDword.dwOutputValue.31);
			(* Exponent *)
			intExponent:=DWORD_TO_INT(SHR(fbConvertWordToDword.dwOutputValue,23) AND 16#FF);
			(* Mantisse *)
			realMantisse:=DWORD_TO_REAL(fbConvertWordToDword.dwOutputValue AND 16#7FFFFF);
			(* Result *)
		str_Data_Out[int_Poll_Count].real_ApparentPower_VA := LREAL_TO_REAL((EXPT((-1),usintSign) * (1+realMantisse/8388608) * EXPT(2,intExponent-127)));
		x:=13;
			fbConvertWordToDword(wInputValue_1:= arrBuffer_FC3[x], wInputValue_2:= arrBuffer_FC3[x+1], eByteOrderForConvert:= eByteOrder.eLittleEndian , dwOutputValue=> );
			(* Sign *)
			usintSign:=BOOL_TO_USINT(fbConvertWordToDword.dwOutputValue.31);
			(* Exponent *)
			intExponent:=DWORD_TO_INT(SHR(fbConvertWordToDword.dwOutputValue,23) AND 16#FF);
			(* Mantisse *)
			realMantisse:=DWORD_TO_REAL(fbConvertWordToDword.dwOutputValue AND 16#7FFFFF);
			(* Result *)
		str_Data_Out[int_Poll_Count].real_Frequency_Hz := LREAL_TO_REAL((EXPT((-1),usintSign) * (1+realMantisse/8388608) * EXPT(2,intExponent-127)));
		x:=41;
			fbConvertWordToDword(wInputValue_1:= arrBuffer_FC3[x], wInputValue_2:= arrBuffer_FC3[x+1], eByteOrderForConvert:= eByteOrder.eLittleEndian , dwOutputValue=> );
			(* Sign *)
			usintSign:=BOOL_TO_USINT(fbConvertWordToDword.dwOutputValue.31);
			(* Exponent *)
			intExponent:=DWORD_TO_INT(SHR(fbConvertWordToDword.dwOutputValue,23) AND 16#FF);
			(* Mantisse *)
			realMantisse:=DWORD_TO_REAL(fbConvertWordToDword.dwOutputValue AND 16#7FFFFF);
			(* Result *)
		str_Data_Out[int_Poll_Count].real_VoltageL1N_V := LREAL_TO_REAL((EXPT((-1),usintSign) * (1+realMantisse/8388608) * EXPT(2,intExponent-127)));
		x:=x+2;
			fbConvertWordToDword(wInputValue_1:= arrBuffer_FC3[x], wInputValue_2:= arrBuffer_FC3[x+1], eByteOrderForConvert:= eByteOrder.eLittleEndian , dwOutputValue=> );
			(* Sign *)
			usintSign:=BOOL_TO_USINT(fbConvertWordToDword.dwOutputValue.31);
			(* Exponent *)
			intExponent:=DWORD_TO_INT(SHR(fbConvertWordToDword.dwOutputValue,23) AND 16#FF);
			(* Mantisse *)
			realMantisse:=DWORD_TO_REAL(fbConvertWordToDword.dwOutputValue AND 16#7FFFFF);
			(* Result *)
		str_Data_Out[int_Poll_Count].real_VoltageL2N_V := LREAL_TO_REAL((EXPT((-1),usintSign) * (1+realMantisse/8388608) * EXPT(2,intExponent-127)));
		x:=x+2;
			fbConvertWordToDword(wInputValue_1:= arrBuffer_FC3[x], wInputValue_2:= arrBuffer_FC3[x+1], eByteOrderForConvert:= eByteOrder.eLittleEndian , dwOutputValue=> );
			(* Sign *)
			usintSign:=BOOL_TO_USINT(fbConvertWordToDword.dwOutputValue.31);
			(* Exponent *)
			intExponent:=DWORD_TO_INT(SHR(fbConvertWordToDword.dwOutputValue,23) AND 16#FF);
			(* Mantisse *)
			realMantisse:=DWORD_TO_REAL(fbConvertWordToDword.dwOutputValue AND 16#7FFFFF);
			(* Result *)
		str_Data_Out[int_Poll_Count].real_VoltageL3N_V := LREAL_TO_REAL((EXPT((-1),usintSign) * (1+realMantisse/8388608) * EXPT(2,intExponent-127)));
		x:=x+2;
			fbConvertWordToDword(wInputValue_1:= arrBuffer_FC3[x], wInputValue_2:= arrBuffer_FC3[x+1], eByteOrderForConvert:= eByteOrder.eLittleEndian , dwOutputValue=> );
			(* Sign *)
			usintSign:=BOOL_TO_USINT(fbConvertWordToDword.dwOutputValue.31);
			(* Exponent *)
			intExponent:=DWORD_TO_INT(SHR(fbConvertWordToDword.dwOutputValue,23) AND 16#FF);
			(* Mantisse *)
			realMantisse:=DWORD_TO_REAL(fbConvertWordToDword.dwOutputValue AND 16#7FFFFF);
			(* Result *)
		str_Data_Out[int_Poll_Count].real_VoltageL1L2_V := LREAL_TO_REAL((EXPT((-1),usintSign) * (1+realMantisse/8388608) * EXPT(2,intExponent-127)));
		x:=x+2;
			fbConvertWordToDword(wInputValue_1:= arrBuffer_FC3[x], wInputValue_2:= arrBuffer_FC3[x+1], eByteOrderForConvert:= eByteOrder.eLittleEndian , dwOutputValue=> );
			(* Sign *)
			usintSign:=BOOL_TO_USINT(fbConvertWordToDword.dwOutputValue.31);
			(* Exponent *)
			intExponent:=DWORD_TO_INT(SHR(fbConvertWordToDword.dwOutputValue,23) AND 16#FF);
			(* Mantisse *)
			realMantisse:=DWORD_TO_REAL(fbConvertWordToDword.dwOutputValue AND 16#7FFFFF);
			(* Result *)
		str_Data_Out[int_Poll_Count].real_VoltageL2L3_V := LREAL_TO_REAL((EXPT((-1),usintSign) * (1+realMantisse/8388608) * EXPT(2,intExponent-127)));
		x:=x+2;
			fbConvertWordToDword(wInputValue_1:= arrBuffer_FC3[x], wInputValue_2:= arrBuffer_FC3[x+1], eByteOrderForConvert:= eByteOrder.eLittleEndian , dwOutputValue=> );
			(* Sign *)
			usintSign:=BOOL_TO_USINT(fbConvertWordToDword.dwOutputValue.31);
			(* Exponent *)
			intExponent:=DWORD_TO_INT(SHR(fbConvertWordToDword.dwOutputValue,23) AND 16#FF);
			(* Mantisse *)
			realMantisse:=DWORD_TO_REAL(fbConvertWordToDword.dwOutputValue AND 16#7FFFFF);
			(* Result *)
		str_Data_Out[int_Poll_Count].real_VoltageL3L1_V := LREAL_TO_REAL((EXPT((-1),usintSign) * (1+realMantisse/8388608) * EXPT(2,intExponent-127)));
		x:=x+2;
			fbConvertWordToDword(wInputValue_1:= arrBuffer_FC3[x], wInputValue_2:= arrBuffer_FC3[x+1], eByteOrderForConvert:= eByteOrder.eLittleEndian , dwOutputValue=> );
			(* Sign *)
			usintSign:=BOOL_TO_USINT(fbConvertWordToDword.dwOutputValue.31);
			(* Exponent *)
			intExponent:=DWORD_TO_INT(SHR(fbConvertWordToDword.dwOutputValue,23) AND 16#FF);
			(* Mantisse *)
			realMantisse:=DWORD_TO_REAL(fbConvertWordToDword.dwOutputValue AND 16#7FFFFF);
			(* Result *)
		str_Data_Out[int_Poll_Count].real_CurrentL1_A := LREAL_TO_REAL((EXPT((-1),usintSign) * (1+realMantisse/8388608) * EXPT(2,intExponent-127)));
		x:=x+2;
			fbConvertWordToDword(wInputValue_1:= arrBuffer_FC3[x], wInputValue_2:= arrBuffer_FC3[x+1], eByteOrderForConvert:= eByteOrder.eLittleEndian , dwOutputValue=> );
			(* Sign *)
			usintSign:=BOOL_TO_USINT(fbConvertWordToDword.dwOutputValue.31);
			(* Exponent *)
			intExponent:=DWORD_TO_INT(SHR(fbConvertWordToDword.dwOutputValue,23) AND 16#FF);
			(* Mantisse *)
			realMantisse:=DWORD_TO_REAL(fbConvertWordToDword.dwOutputValue AND 16#7FFFFF);
			(* Result *)
		str_Data_Out[int_Poll_Count].real_CurrentL2_A := LREAL_TO_REAL((EXPT((-1),usintSign) * (1+realMantisse/8388608) * EXPT(2,intExponent-127)));
		x:=x+2;
			fbConvertWordToDword(wInputValue_1:= arrBuffer_FC3[x], wInputValue_2:= arrBuffer_FC3[x+1], eByteOrderForConvert:= eByteOrder.eLittleEndian , dwOutputValue=> );
			(* Sign *)
			usintSign:=BOOL_TO_USINT(fbConvertWordToDword.dwOutputValue.31);
			(* Exponent *)
			intExponent:=DWORD_TO_INT(SHR(fbConvertWordToDword.dwOutputValue,23) AND 16#FF);
			(* Mantisse *)
			realMantisse:=DWORD_TO_REAL(fbConvertWordToDword.dwOutputValue AND 16#7FFFFF);
			(* Result *)
		str_Data_Out[int_Poll_Count].real_CurrentL3_A := LREAL_TO_REAL((EXPT((-1),usintSign) * (1+realMantisse/8388608) * EXPT(2,intExponent-127)));
		x:=65;
			fbConvertWordToDword(wInputValue_1:= arrBuffer_FC3[x], wInputValue_2:= arrBuffer_FC3[x+1], eByteOrderForConvert:= eByteOrder.eLittleEndian , dwOutputValue=> );
			(* Sign *)
			usintSign:=BOOL_TO_USINT(fbConvertWordToDword.dwOutputValue.31);
			(* Exponent *)
			intExponent:=DWORD_TO_INT(SHR(fbConvertWordToDword.dwOutputValue,23) AND 16#FF);
			(* Mantisse *)
			realMantisse:=DWORD_TO_REAL(fbConvertWordToDword.dwOutputValue AND 16#7FFFFF);
			(* Result *)
		str_Data_Out[int_Poll_Count].real_EnergyperDay_Wh := LREAL_TO_REAL((EXPT((-1),usintSign) * (1+realMantisse/8388608) * EXPT(2,intExponent-127)));
		x:=x+2;
			fbConvertWordToDword(wInputValue_1:= arrBuffer_FC3[x], wInputValue_2:= arrBuffer_FC3[x+1], eByteOrderForConvert:= eByteOrder.eLittleEndian , dwOutputValue=> );
			(* Sign *)
			usintSign:=BOOL_TO_USINT(fbConvertWordToDword.dwOutputValue.31);
			(* Exponent *)
			intExponent:=DWORD_TO_INT(SHR(fbConvertWordToDword.dwOutputValue,23) AND 16#FF);
			(* Mantisse *)
			realMantisse:=DWORD_TO_REAL(fbConvertWordToDword.dwOutputValue AND 16#7FFFFF);
			(* Result *)
		str_Data_Out[int_Poll_Count].real_EnergyTotal_Wh := LREAL_TO_REAL((EXPT((-1),usintSign) * (1+realMantisse/8388608) * EXPT(2,intExponent-127)));
		iStateModbusRead := 4;
	4://Wait and go to step 1
		//1 because 0 is the Init Step for Read
		timer_Wait.IN := TRUE;
		
		IF timer_Wait.Q = TRUE THEN
			iStateModbusRead := 1;
			timer_Wait.IN :=FALSE;
		END_IF

			
		
		//Error on Master, changes on Inputs or Timeout
		IF timer_Timeout.Q THEN 
			iStateModbusError := 300; 
		END_IF
		

	
END_CASE

(* wait timer*)

timer_Wait(PT:=T#3S);


(*------------------------------------------------------------------Error and Warning----------------------------------------------------------------------------*)	
 
timer_Connection_ok			(In:=int_Data_Received<>int_Data_Received_old,PT:=T#10S);
timer_Connection_ok_TOF		(In:=NOT(int_Data_Received<>int_Data_Received_old) AND int_Data_Received>3 ,PT:=T#20S);
int_Data_Received_old:=int_Data_Received;
str_Data_Out[int_Poll_Count].m_PollSuccessful:=NOT timer_Connection_ok.Q AND timer_Connection_ok_TOF.Q ;

(*------------------------------------------------------------------------------------------Modbus TCP Functions---------------------------------------------------------------------------------------------*)

fbMBRead_FC3(	sIPAddr:= str_IPAdress, 
				nTCPPort:= 502,
				cbLength:= SIZEOF(arrBuffer_FC3), 
				pDestAddr:= ADR(arrBuffer_FC3), 
				tTimeout:= T#10S,
				nErrId => str_Data_Out[int_Poll_Count].udint_Error_ID);

				
FPError_FC_3(CLK:= fbMBRead_FC3.bError, Q=> );		

(*------------------------------------------------------------------------------------------State Machine Error---------------------------------------------------------------------------------------------*)	

CASE iStateModbusError OF
	
	300://Error
		timer_Wait.IN :=TRUE;
		timer_Delay.IN := FALSE;
		fbMBRead_FC3.bExecute := FALSE;
		m_MBTCPError := TRUE; 		
		m_Poll_ok:=FALSE;
		int_Data_Received:=0;
				//Restart from new with the Read out part after an Error
		IF timer_Wait.Q = TRUE THEN
			iStateModbusRead := 0;	
			iStateModbusError := 0;
			timer_Wait.IN :=FALSE;
			timer_Timeout.IN := FALSE;
		END_IF		
							
END_CASE

END_FUNCTION_BLOCK

// ---- FBs/PhoenixContact/FB_PhoenixContact_EM_EEM_EM375.TcPOU
FUNCTION_BLOCK FB_PhoenixContact_EM_EEM_EM375
VAR_INPUT PERSISTENT
	///Enable the function
	bEnable: BOOL;
	///Unit ID
	byUnitID: BYTE := 1;
	///IP Adress from the Meter					
	sIPAdress: STRING(15);
END_VAR
VAR_OUTPUT
	///Output structure with Data from Electric Meter (Power Data)
	stDataEMPower: ST_ElectricMeter_Output_Power;
	///Output structure with Data from Electric Meter (Counter Data)
	stDataEMCounter: ST_ElectricMeter_Output_Counter;
	///Output structure with Data from Electric Meter (Power Data RealTime)
	stDataEMPowerRealTime: ST_ElectricMeter_Output_Power;
	///Output structure with Data from Electric Meter (Counter Data RealTime)
	stDataEMCounterRealTime: ST_ElectricMeter_Output_Counter;
	///Active Number from the Electric Meter for using on other functions
	diNrOfEM_OUT: DINT;
END_VAR
VAR
	///Electric Meter Function
	{attribute 'conditionalshow' := ''}
	fbEM: FB_ElectricMeter;
	///Function block to calcualte the number of the Device
	{attribute 'hide' := ''}
	fbNumberDevice: FB_NumberOfDevice;
	///Modbus Read Function (FC3)
	{attribute 'hide' := ''}
	fbMBRead_FC3: FB_MBReadRegs;
	///Convert function
	{attribute 'hide' := ''}
	fbConvertData: FB_CV_WORD_TO_DWORD;
	///Timer to dissable the Function after Lynus_Standards.Constants_General.tTimeDissableLynusFunctions Days without connection to the Lynus Cloud
	{attribute 'hide' := ''}
	timDissableFunctions: TON;
	///Timer to try reset the connection Flag on the GVL. (When somebody delete the Connection Function and make only a onlinechange)
	{attribute 'hide' := ''}
	timResetConnectionOnGVL: TON;
	///Timer for Delay between Requests
	{attribute 'hide' := ''}
	timDelay: TON;
	///Timer for Timeout
	{attribute 'hide' := ''}
	timTimeout: TON;
	///Timer to Close the Socket after to much Errors
	{attribute 'hide' := ''}
	timCloseSocket: TON;
	///Internal positive Edge
	{attribute 'hide' := ''}
	FPEnable: R_TRIG;
	///Internal positive Edge
	{attribute 'hide' := ''}
	FPError_FC_3: R_TRIG;
	///Function to save persistent data
	{attribute 'hide' := ''}
	PD_String: FB_PersistentData_String;
	///Function to save persistent data
	{attribute 'hide' := ''}
	arrPD: ARRAY[1..2] OF FB_PersistentData_Number;
	///Buffer with Data from FC3
	{attribute 'hide' := ''}
	arrBuffer_FC3: ARRAY[1..62] OF WORD;
	///Error from Table A-17
	{attribute 'hide' := ''}
	bErrorFromDevice: BOOL;
	///Wait in Step before start to clean data on PLC
	{attribute 'hide' := ''}
	byWaitInStep: BYTE;
	///Modbus TCP Function Error	Counter
	{attribute 'hide' := ''}
	byMBTCPErrorCounter: BYTE;
	///State machine to handle the data on the GVL
	{attribute 'hide' := ''}
	iStateGVLData: INT;
	///State variable for Statemachine
	{attribute 'hide' := ''}
	iStateModbusRead: INT;
	///State variable for Statemachine
	{attribute 'hide' := ''}
	iStateModbusError: INT;
	///Compare State variable
	{attribute 'hide' := ''}
	iStateModbus_CP: INT;
	///Counter to clean old data on GVL
	{attribute 'hide' := ''}
	diCounterForGVL: DINT;
END_VAR

//Creator : Kai Ebensperger
//Company : Lynus AG
//Date : 19.09.2021
//Version : 1.0.0.0

//With this function block its possible to read out a Electric Meter EEM-EM375 from the Factory Phönix Contact.
//This Function Block read out the Default Values from the Electric Meter from Table A-2 and Table A-3 and Table A-17 for Errormessage
//Version according to which was implemented : Revision 00

//NOTE for diNr.....Designation => 
//_IN = Here Data come in from other Functions or go out to other functions about the GVL
//_OUT = Here Data go out to other functions about the GVL

(*-------------------------------------------------------------Calcualte the number of EM---------------------------------------------------------------*)

fbNumberDevice(
	diActualNumberOfDevices:= Lynus_Standards.GVL_Energy.stNumberOfDevices.diNumberOfElectricMeters, 
	diMaxNumberOfDevices:= Constants_Energy.diMaxNumberOfElectricMeters, 
	udiCounterOnlineChange:= TwinCAT_SystemInfoVarList._AppInfo.OnlineChangeCnt, 
	bNumberIsCalculatet=> , 
	bFPNumberIsCalculatet=> , 
	bOnlineChange=> , 
	diNumberForThisDevice=> diNrOfEM_OUT, 
	diNumberOfTotalDevices=> );

//Write new Numer on GVL
IF fbNumberDevice.bFPNumberIsCalculatet THEN
	Lynus_Standards.GVL_Energy.stNumberOfDevices.diNumberOfElectricMeters := fbNumberDevice.diNumberOfTotalDevices;	
END_IF

//Delete old Number on GVL
IF fbNumberDevice.bOnlineChange THEN 
	Lynus_Standards.GVL_Energy.stNumberOfDevices.diNumberOfElectricMeters := diNrOfEM_OUT;	
		iStateGVLData := 1; 
END_IF

(*-------------------------------------------------------------Service from Backend is ready and check the connection to backen for dissabel/enable Function---------------------------------------------------------------*)

//Try to reset the variable for connection on the GVL. When all is normal then the Lynus Mqtt connection function set this variable to true in the next cycle
//When we have no connection to the backend then after Lynus_Standards.Constants_General.tTimeDissableLynusFunctions days the Function is dissabled with all of his functionalities
timResetConnectionOnGVL(IN:= NOT timResetConnectionOnGVL.Q, PT:= T#1H, Q=> , ET=> );
	IF timResetConnectionOnGVL.Q THEN Lynus_Standards.GVL_Communicator.bStateConnectionToEnableFunctions := FALSE; END_IF
		IF NOT Lynus_Standards.GVL_Communicator.bStateConnectionToEnableFunctions THEN timDissableFunctions.IN := TRUE; ELSE timDissableFunctions.IN := FALSE; END_IF  
			timDissableFunctions(IN:= , PT:= Lynus_Standards.Constants_General.tTimeDissableLynusFunctions, Q=> , ET=> );

(*------------------------------------------------------------------------------------------State Machine Read---------------------------------------------------------------------------------------------*)

//Start the Statemachine
FPEnable(CLK:= bEnable, Q=> );
	IF FPEnable.Q AND iStateModbusRead = 0 AND iStateModbusRead = 0 AND iStateModbusError = 0 THEN 
			iStateModbusRead := 1; 
	END_IF
		IF NOT bEnable THEN iStateModbusRead := 0; iStateModbusError := 0; END_IF

//Timer for delay
timDelay(IN:= , PT:= T#150MS, Q=> , ET=> );

//Timer for Timeout in Statemachine
IF iStateModbusRead > 0 AND iStateModbusRead <= 2 AND iStateModbusRead = iStateModbus_CP THEN
		timTimeout.IN := TRUE;
ELSE	
		timTimeout.IN := FALSE;
END_IF 
	IF iStateModbusRead = 0 THEN timTimeout.IN := FALSE; END_IF
		timTimeout(IN:= , PT:= T#20S, Q=> , ET=> );			
			
CASE iStateModbusRead OF
	
	0://Init State
		iStateModbus_CP := 0;
			timDelay.IN := FALSE;
				fbMBRead_FC3.bExecute := FALSE;

	1://Read out Table A-2
		iStateModbus_CP := iStateModbusRead;
		
		fbMBRead_FC3.nQuantity := 62;
			fbMBRead_FC3.nMBAddr := 50512;
				fbMBRead_FC3.bExecute := TRUE;
					fbMBRead_FC3.nUnitID := byUnitID;
			
		IF fbMBRead_FC3.bBusy THEN timDelay.IN := TRUE; END_IF
		
		//Wait for Delay, copy Data and then next step
		IF NOT fbMBRead_FC3.bBusy AND NOT fbMBRead_FC3.bError AND timDelay.Q THEN
			//Actual Values from Meter form Table A-2
			fbConvertData(wInputValue_1:= arrBuffer_FC3[3], wInputValue_2:= arrBuffer_FC3[4], eByteOrderForConvert:= eByteOrder.eBigEndian, dwOutputValue=> );
				fbEM.lrVoltageL1L2 := DWORD_TO_LREAL(fbConvertData.dwOutputValue) / 100;
			fbConvertData(wInputValue_1:= arrBuffer_FC3[5], wInputValue_2:= arrBuffer_FC3[6], eByteOrderForConvert:= eByteOrder.eBigEndian, dwOutputValue=> );
				fbEM.lrVoltageL2L3 := DWORD_TO_LREAL(fbConvertData.dwOutputValue) / 100;
			fbConvertData(wInputValue_1:= arrBuffer_FC3[7], wInputValue_2:= arrBuffer_FC3[8], eByteOrderForConvert:= eByteOrder.eBigEndian, dwOutputValue=> );
				fbEM.lrVoltageL3L1 := DWORD_TO_LREAL(fbConvertData.dwOutputValue) / 100;
			fbConvertData(wInputValue_1:= arrBuffer_FC3[9], wInputValue_2:= arrBuffer_FC3[10], eByteOrderForConvert:= eByteOrder.eBigEndian, dwOutputValue=> );
				fbEM.lrVoltageL1N := DWORD_TO_LREAL(fbConvertData.dwOutputValue) / 100;
			fbConvertData(wInputValue_1:= arrBuffer_FC3[11], wInputValue_2:= arrBuffer_FC3[12], eByteOrderForConvert:= eByteOrder.eBigEndian, dwOutputValue=> );
				fbEM.lrVoltageL2N := DWORD_TO_LREAL(fbConvertData.dwOutputValue) / 100;
			fbConvertData(wInputValue_1:= arrBuffer_FC3[13], wInputValue_2:= arrBuffer_FC3[14], eByteOrderForConvert:= eByteOrder.eBigEndian, dwOutputValue=> );
				fbEM.lrVoltageL3N := DWORD_TO_LREAL(fbConvertData.dwOutputValue) / 100;	
			fbConvertData(wInputValue_1:= arrBuffer_FC3[15], wInputValue_2:= arrBuffer_FC3[16], eByteOrderForConvert:= eByteOrder.eBigEndian, dwOutputValue=> );
				fbEM.lrFrequency := DWORD_TO_LREAL(fbConvertData.dwOutputValue) / 100;
			fbConvertData(wInputValue_1:= arrBuffer_FC3[17], wInputValue_2:= arrBuffer_FC3[18], eByteOrderForConvert:= eByteOrder.eBigEndian, dwOutputValue=> );
				fbEM.lrCurrentL1 := DWORD_TO_LREAL(fbConvertData.dwOutputValue) / 1000;				
			fbConvertData(wInputValue_1:= arrBuffer_FC3[19], wInputValue_2:= arrBuffer_FC3[20], eByteOrderForConvert:= eByteOrder.eBigEndian, dwOutputValue=> );
				fbEM.lrCurrentL2 := DWORD_TO_LREAL(fbConvertData.dwOutputValue) / 1000;	
			fbConvertData(wInputValue_1:= arrBuffer_FC3[21], wInputValue_2:= arrBuffer_FC3[22], eByteOrderForConvert:= eByteOrder.eBigEndian, dwOutputValue=> );
				fbEM.lrCurrentL3 := DWORD_TO_LREAL(fbConvertData.dwOutputValue) / 1000;		
			fbConvertData(wInputValue_1:= arrBuffer_FC3[25], wInputValue_2:= arrBuffer_FC3[26], eByteOrderForConvert:= eByteOrder.eBigEndian, dwOutputValue=> );
				fbEM.lrPowerTotal := DINT_TO_LREAL(DWORD_TO_DINT(fbConvertData.dwOutputValue)) / 0.1;		
			fbConvertData(wInputValue_1:= arrBuffer_FC3[27], wInputValue_2:= arrBuffer_FC3[28], eByteOrderForConvert:= eByteOrder.eBigEndian, dwOutputValue=> );
				fbEM.lrReactivePowerTotal := DINT_TO_LREAL(DWORD_TO_DINT(fbConvertData.dwOutputValue)) / 0.1;				
			fbConvertData(wInputValue_1:= arrBuffer_FC3[29], wInputValue_2:= arrBuffer_FC3[30], eByteOrderForConvert:= eByteOrder.eBigEndian, dwOutputValue=> );
				fbEM.lrApparentPowerTotal := DWORD_TO_LREAL(fbConvertData.dwOutputValue) / 0.1;
			fbConvertData(wInputValue_1:= arrBuffer_FC3[33], wInputValue_2:= arrBuffer_FC3[34], eByteOrderForConvert:= eByteOrder.eBigEndian, dwOutputValue=> );
				fbEM.lrPowerL1 := DINT_TO_LREAL(DWORD_TO_DINT(fbConvertData.dwOutputValue)) / 0.1;
			fbConvertData(wInputValue_1:= arrBuffer_FC3[35], wInputValue_2:= arrBuffer_FC3[36], eByteOrderForConvert:= eByteOrder.eBigEndian, dwOutputValue=> );
				fbEM.lrPowerL2 := DINT_TO_LREAL(DWORD_TO_DINT(fbConvertData.dwOutputValue)) / 0.1;				
			fbConvertData(wInputValue_1:= arrBuffer_FC3[37], wInputValue_2:= arrBuffer_FC3[38], eByteOrderForConvert:= eByteOrder.eBigEndian, dwOutputValue=> );
				fbEM.lrPowerL3 := DINT_TO_LREAL(DWORD_TO_DINT(fbConvertData.dwOutputValue)) / 0.1;	
				
			//Next Step
			fbMBRead_FC3.bExecute := FALSE;
				timDelay.IN := FALSE;
					iStateModbusRead := 2;
		END_IF
		
		//Error or Timeout
		IF FPError_FC_3.Q OR timTimeout.Q THEN
			iStateModbusError := 300;
				iStateModbusRead := - 1;
		END_IF
	
	2://Read out Table A-3
		iStateModbus_CP := iStateModbusRead;
		
		fbMBRead_FC3.nQuantity := 22;
			fbMBRead_FC3.nMBAddr := 50768;
				fbMBRead_FC3.bExecute := TRUE;
					fbMBRead_FC3.nUnitID := byUnitID;
			
		IF fbMBRead_FC3.bBusy THEN timDelay.IN := TRUE; END_IF
		
		//Wait for Delay, copy Data and then next step
		IF NOT fbMBRead_FC3.bBusy AND NOT fbMBRead_FC3.bError AND timDelay.Q THEN
			//Counters from Meter form Table A-3
			fbConvertData(wInputValue_1:= arrBuffer_FC3[3], wInputValue_2:= arrBuffer_FC3[4], eByteOrderForConvert:= eByteOrder.eBigEndian, dwOutputValue=> );
				fbEM.lrCounterEnergyT1_Consumption := DWORD_TO_LREAL(fbConvertData.dwOutputValue);
					fbEM.lrTotalCounterEnergy_Consumption := fbEM.lrCounterEnergyT1_Consumption;
			fbConvertData(wInputValue_1:= arrBuffer_FC3[9], wInputValue_2:= arrBuffer_FC3[10], eByteOrderForConvert:= eByteOrder.eBigEndian, dwOutputValue=> );
				fbEM.lrCounterEnergyT1_Production := DWORD_TO_LREAL(fbConvertData.dwOutputValue);
					fbEM.lrTotalCounterEnergy_Production := fbEM.lrCounterEnergyT1_Production;
				
			//Next Step
			fbMBRead_FC3.bExecute := FALSE;
				timDelay.IN := FALSE;
					iStateModbusRead := 3;
		END_IF
		
		//Error or Timeout
		IF FPError_FC_3.Q OR timTimeout.Q THEN
			iStateModbusError := 300;
				iStateModbusRead := - 1;
		END_IF		
		
	3://Read out Table A-17
		iStateModbus_CP := iStateModbusRead;
		
		fbMBRead_FC3.nQuantity := 2;
			fbMBRead_FC3.nMBAddr := 1300;
				fbMBRead_FC3.bExecute := TRUE;
					fbMBRead_FC3.nUnitID := byUnitID;
			
		IF fbMBRead_FC3.bBusy THEN timDelay.IN := TRUE; END_IF
		
		//Wait for Delay, copy Data and then next step
		IF NOT fbMBRead_FC3.bBusy AND NOT fbMBRead_FC3.bError AND timDelay.Q THEN
			//Meter Error Message form Table A-17
			fbConvertData(wInputValue_1:= arrBuffer_FC3[1], wInputValue_2:= arrBuffer_FC3[2], eByteOrderForConvert:= eByteOrder.eBigEndian, dwOutputValue=> );
				IF fbConvertData.dwOutputValue <> 0 THEN bErrorFromDevice := TRUE; ELSE bErrorFromDevice := FALSE; END_IF  
				
			//Next Step
			fbMBRead_FC3.bExecute := FALSE;
				timDelay.IN := FALSE;
					iStateModbusRead := 1;
		END_IF
		
		//Error or Timeout
		IF FPError_FC_3.Q OR timTimeout.Q THEN
			iStateModbusError := 300;
				iStateModbusRead := - 1;
		END_IF
		
END_CASE

(*----------------------------------------------------------------------------------------Electric Meter Function----------------------------------------------------------------------------------------------*)

//Error
IF timDissableFunctions.Q THEN fbEM.bWarning := TRUE; fbEM.iWarningCode := 0; ELSE fbEM.bWarning := FALSE; END_IF 
	IF Lynus_Standards.GVL_Energy.stNumberOfDevices.diNumberOfElectricMeters > Constants_Energy.diMaxNumberOfElectricMeters OR byMBTCPErrorCounter > 10 OR bErrorFromDevice THEN fbEM.bError := TRUE; ELSE fbEM.bError := FALSE; END_IF
		IF Lynus_Standards.GVL_Energy.stNumberOfDevices.diNumberOfElectricMeters > Constants_Energy.diMaxNumberOfElectricMeters THEN fbEM.iErrorCode := 1;
		ELSIF  byMBTCPErrorCounter > 10 OR bErrorFromDevice THEN fbEM.iErrorCode := 0;
		END_IF

IF iStateModbusRead <> 2 THEN fbEM.bReadOutDataDone := TRUE; ELSE fbEM.bReadOutDataDone := FALSE; END_IF  		
		
//Function
fbEM(
	bEnable:= bEnable AND NOT timDissableFunctions.Q, 
	bError:= , 
	bEnableReadOutFunction:= FALSE, 
	bWriteWithDelay:= TRUE, 
	bPowerDataInvers:= FALSE,
	bReadOutDataDone:= ,
	iTimeReadOutInterval:= 0, 
	iErrorCode:= , 
	iWarningCode:= , 
	lrTotalCounterEnergy_Consumption:= , 
	lrTotalCounterEnergy_Production:= , 
	lrCounterEnergyT1_Consumption:= , 
	lrCounterEnergyT2_Consumption:= 0, 
	lrCounterEnergyT1_Production:= , 
	lrCounterEnergyT2_Production:= 0, 
	lrCurrentL1:= , 
	lrVoltageL1N:= , 
	lrVoltageL1L2:= , 
	lrPowerL1:= , 
	lrCurrentL2:= , 
	lrVoltageL2N:= , 
	lrVoltageL2L3:= , 
	lrPowerL2:= , 
	lrCurrentL3:= , 
	lrVoltageL3N:= , 
	lrVoltageL3L1:= , 
	lrPowerL3:= , 
	lrPowerTotal:= , 
	lrFrequency:= , 
	lrReactivePowerTotal:= , 
	lrApparentPowerTotal:= , 
	tTimDelayOutput:= T#5S, 
	stDataEMOutPower=> stDataEMPowerRealTime, 
	stDataEMOutPowerDelay=> stDataEMPower, 
	stDataEMOutCounter=> stDataEMCounterRealTime,
	stDataEMOutCounterDelay=> stDataEMCounter,
	bReadOutMeter=> );

(*------------------------------------------------------------------------------------------State Machine Error---------------------------------------------------------------------------------------------*)	

CASE iStateModbusError OF
	
	300://Error
		iStateModbus_CP := iStateModbusError;
			timDelay.IN := FALSE;
				fbMBRead_FC3.bExecute := FALSE;
					byMBTCPErrorCounter := byMBTCPErrorCounter + 1;
						byMBTCPErrorCounter := LIMIT(0,byMBTCPErrorCounter,11);
							//Restart from new with the Read out part after an Error
							IF byMBTCPErrorCounter < 10 THEN
								iStateModbusRead := 1;	
									iStateModbusError := 0;
							ELSE
								//Wait here in the Error State for the Delay Timer and then we dont have a Timeout Error
								iStateModbusRead := - 1;
									//Start from New when the Delay is paste
									IF timCloseSocket.Q THEN
										iStateModbusRead := 1;	
											iStateModbusError := 0;
												byMBTCPErrorCounter := 0;
									END_IF
							END_IF
						
END_CASE

//Timer to close the Socket after to much TCP Errors and reopen a new one
timCloseSocket(IN:= byMBTCPErrorCounter > 10 AND bEnable, PT:= T#1M, Q=> , ET=> );

(*------------------------------------------------------------------------------------------Modbus TCP Functions---------------------------------------------------------------------------------------------*)

fbMBRead_FC3(sIPAddr:= sIPAdress, nTCPPort:= 502, nUnitID := byUnitID, cbLength:= SIZEOF(arrBuffer_FC3), pDestAddr:= ADR(arrBuffer_FC3), tTimeout:= T#2S );
	FPError_FC_3(CLK:= fbMBRead_FC3.bError, Q=> );
	
(*-----------------------------------------------------------Handle data to Global structure for Electric Meter-----------------------------------------------------------------*)

CASE iStateGVLData OF
	
	0://Init Step
		byWaitInStep := 0;
			diCounterForGVL := 1;
	
	1://Wait for 4 Steps before clean al Data on GVL
		byWaitInStep := byWaitInStep + 1;
			IF byWaitInStep >= 4 AND fbNumberDevice.bNumberIsCalculatet THEN iStateGVLData := 2; END_IF
				//To much Devices, back to the Init step
				IF byWaitInStep >= 4 AND NOT fbNumberDevice.bNumberIsCalculatet THEN iStateGVLData := 0; END_IF	
			
	2://Clear all Data in GVL
		Lynus_Standards.GVL_Energy.stDataElectricMeters[diCounterForGVL].bEnabled := FALSE;	
			Lynus_Standards.GVL_Energy.stDataElectricMeters[diCounterForGVL].byErrorWarning := 0;
				Lynus_Standards.GVL_Energy.stDataElectricMeters[diCounterForGVL].lrCounterEnergyT1_Consumption := 0;
					Lynus_Standards.GVL_Energy.stDataElectricMeters[diCounterForGVL].lrCounterEnergyT1_Production := 0;
						Lynus_Standards.GVL_Energy.stDataElectricMeters[diCounterForGVL].lrCounterEnergyT2_Consumption := 0;
							Lynus_Standards.GVL_Energy.stDataElectricMeters[diCounterForGVL].lrCounterEnergyT2_Production := 0;
								Lynus_Standards.GVL_Energy.stDataElectricMeters[diCounterForGVL].lrPower := 0;
									Lynus_Standards.GVL_Energy.stDataElectricMeters[diCounterForGVL].lrPowerConsumption := 0;
										Lynus_Standards.GVL_Energy.stDataElectricMeters[diCounterForGVL].lrPowerProduction := 0;
											Lynus_Standards.GVL_Energy.stDataElectricMeters[diCounterForGVL].lrTotalCounterEnergy_Consumption := 0;
												Lynus_Standards.GVL_Energy.stDataElectricMeters[diCounterForGVL].lrTotalCounterEnergy_Production := 0;
		
		//Electric Meters
		diCounterForGVL := diCounterForGVL + 1;
			diCounterForGVL := LIMIT(0,diCounterForGVL,Constants_Energy.diMaxNumberOfElectricMeters);
				//Back to the init step
				IF diCounterForGVL >= Constants_Energy.diMaxNumberOfElectricMeters THEN iStateGVLData := 0; END_IF

END_CASE 	 

//Write Data on GVL for Electric Meter
IF diNrOfEM_OUT > 0 AND fbNumberDevice.bNumberIsCalculatet THEN
	Lynus_Standards.GVL_Energy.stDataElectricMeters[diNrOfEM_OUT].bEnabled := fbEM.stDataEMOutPower.bEnabled;
		Lynus_Standards.GVL_Energy.stDataElectricMeters[diNrOfEM_OUT].byErrorWarning := fbEM.stDataEMOutPower.byErrorWarning;
			Lynus_Standards.GVL_Energy.stDataElectricMeters[diNrOfEM_OUT].lrCounterEnergyT1_Consumption := fbEM.stDataEMOutCounter.lrCounterEnergyT1_Consumption;
				Lynus_Standards.GVL_Energy.stDataElectricMeters[diNrOfEM_OUT].lrCounterEnergyT1_Production := fbEM.stDataEMOutCounter.lrCounterEnergyT1_Production;
					Lynus_Standards.GVL_Energy.stDataElectricMeters[diNrOfEM_OUT].lrCounterEnergyT2_Consumption := fbEM.stDataEMOutCounter.lrCounterEnergyT2_Consumption;
						Lynus_Standards.GVL_Energy.stDataElectricMeters[diNrOfEM_OUT].lrCounterEnergyT2_Production := fbEM.stDataEMOutCounter.lrCounterEnergyT2_Production;		
							Lynus_Standards.GVL_Energy.stDataElectricMeters[diNrOfEM_OUT].lrPower := fbEM.stDataEMOutPower.lrPowerTotal;
								Lynus_Standards.GVL_Energy.stDataElectricMeters[diNrOfEM_OUT].lrPowerConsumption := fbEM.stDataEMOutPower.lrPowerConsumption;
									Lynus_Standards.GVL_Energy.stDataElectricMeters[diNrOfEM_OUT].lrPowerProduction := fbEM.stDataEMOutPower.lrPowerProduction;
										Lynus_Standards.GVL_Energy.stDataElectricMeters[diNrOfEM_OUT].lrTotalCounterEnergy_Consumption := fbEM.stDataEMOutCounter.lrTotalCounterEnergy_Consumption;
											Lynus_Standards.GVL_Energy.stDataElectricMeters[diNrOfEM_OUT].lrTotalCounterEnergy_Production := fbEM.stDataEMOutCounter.lrTotalCounterEnergy_Production;
END_IF

(*----------------------------------------------------------Save persistent data----------------------------------------------------------------*)

arrPD[1](lrValue:= BOOL_TO_LREAL(bEnable), bEventBasedActive=> );
arrPD[2](lrValue:= BYTE_TO_LREAL(byUnitID), bEventBasedActive=> );
PD_String(sText:= sIPAdress, bEventBasedActive=> );

END_FUNCTION_BLOCK

// ---- FBs/Pixii/FB_Pixii_v1.TcPOU
FUNCTION_BLOCK FB_Pixii_v1
VAR_INPUT PERSISTENT
	bEnable							: BOOL;											//{#lynus.ag#()} //True = Function is enabled, FALSE = Function is dissabled, no new Data
	bActivateControl				: BOOL;											//Activate the control  over Modbus TCP (False = Inverter work by himself)
	byUnitID						: BYTE:=1;										//Unit ID fromt the Inverter (0 to 255)
	byPriority						: BYTE;											//{#lynus.ag#()} //Priority of the Device
	diNrOfEMS_IN					: DINT;											//Number of EMS what control this Device.
	lrMaxCapacityBattery			: LREAL;										//{#lynus.ag#()} //Max Capacity from the Battery in kWh. Here on this Function this Input Value cames from Inside of the Function.
	sIPAdress						: STRING(15);									//IP Adress from the Inverter
END_VAR
VAR_INPUT
	bReset							: BOOL;											//{#lynus.ag#()} //Reset the device after a Error or a Warning
	m_ManualSetpointEnable			: BOOL;											// enable the manual setpoint operation
	i_SetpointPower_Manual_kW		: INT;											// Battery Setpoint, for testing purpose *100=[W]
	m_ManualChargeDischargeMax		: BOOL;											// Enable max charge/Discharge power instead of storage read out vaules
	r_MaxChargePower_W				: REAL;											// max charge power in [W]
	r_MaxDischargePower_W			: REAL;											// max discharge power in [W]
	
END_VAR
VAR_OUTPUT
	stDataPixii						: ST_Pixii_OutData;								//Shows the specific output data from the Xelectric device
	stDataBatt						: ST_Battery_Output;							//{#lynus.ag#()} //Output structure with Data from Battery
	stDataBattInverter				: ST_BatteryInverter_Output;					//{#lynus.ag#()} //Output structure with Data from Battery Inverter
	stDataEMPower					: ST_ElectricMeter_Output_Power;				//Output structure with Data from Electric Meter Grid (Power Data)
	stDataEMCounter					: ST_ElectricMeter_Output_Counter;				//Output structure with Data from Electric Meter Grid (Counter Data)
	diNrOfBatt_OUT					: DINT;											//Active Number from the Battery Function for using on other functions
	diNrOfBattInverter_OUT			: DINT;											//Active Number from the Battery Inverter Function for using on other functions
	diNrOfEM_OUT_Grid				: DINT;											//Active Number from the Electric Meter for using on other functions
	lrMaxCapacityBattery_OUT		: LREAL;										//Max kWh from the Battery system. The Pixii System deliver this value.
	iSetpointPower_Info				: INT;											// Battery Setpoint, for monitoring purpose
END_VAR
VAR
	
	fbBattery						: FB_Battery;									//Function block for battery
	
	fbBatteryInverter				: FB_BatteryInverter;							//Function block for battery inveter
	
	fbEMPower						: FB_ElectricMeter;								//Electric Meter Function 
	
	fbPIDChrgStandby				: FB_PID;										//Controller to control the battery current on 0 in the standby mode	
	
	fbNumberDeviceBattery			: FB_NumberOfDevice;							//Function block to calcualte the number of the Device
	
	fbNumberDeviceBatteryInvert		: FB_NumberOfDevice;							//Function block to calcualte the number of the Device
	
	fbNumberDeviceGrid				: FB_NumberOfDevice;							//Function block to calcualte the number of the Device
	
	fbMBRead_FC3					: FB_MBReadRegs;								//Modbus Read Function (FC3)
	
	fbMBWrite_FC6					: FB_MBWriteSingleReg;								//Modbus Write Function (FC6)
	
	fbConvertData					: FB_CV_WORD_TO_DWORD;							//Convert 2 Words in a Dword
	
	timDelay						: TON;											//Timer for Delay between Requests
	
	timTimeout						: TON;											//Timer for Timeout
	
	timDissableFunctions			: TON;											//Timer to dissable the Function after Lynus_Standards.Constants_General.tTimeDissableLynusFunctions Days without connection to the Lynus Cloud
	
	timResetConnectionOnGVL			: TON;											//Timer to try reset the connection Flag on the GVL. (When somebody delete the Connection Function and make only a onlinechange)
	
	timReset						: TON;											//Timer to reset the Inverter after a Error
	
	timErrorMTCP					: TON;											//Delay when Error on Modbus TCP
	
	timSetStandbyCntrl				: TOF;											//Timer to set the Standby Controller
	
	FPEnable						: R_TRIG;										//Internal positive Edge
	
	FPError_FC_3					: R_TRIG;										//Internal positive Edge
	
	FPError_FC_6					: R_TRIG;										//Internal positive Edge
	
	FPActivateControl				: R_TRIG;										//Internal positive Edge
	
	FNTimDissable					: F_TRIG;										//Internal negative Edge
	
	PD_String						: FB_PersistentData_String;						//Function to save persistent data
	
	arrPD							: ARRAY[1..7] OF FB_PersistentData_Number;		//Function to save persistent data
	
	arrBuffer_FC3					: ARRAY[1..125] OF WORD;							//Buffer with Data from FC3
	
	wordBuffer_FC6					: WORD;								//Buffer with Data from FC16
	
	arrCounterForGVL				: ARRAY[1..3] OF DINT;							//Counter to clean old data on GVL
	
	bEnergyGridConsReceived			: BOOL;											//Energy Consumption from Grid first time received
	
	bEnergyGridProdReceived			: BOOL;											//Energy Production from Grid first time received
	
	byWaitInStep					: BYTE;											//Wait in Step before start to clean data on PLC
	
	byLPWorkAroundACDevice			: BYTE;											//Loop for Workaround
	
//	byNumberOfZero					: BYTE;											//Number with 0 Value from AC Messurement
	
	iSetpointPower					: INT;											//Power Setpoint in W
	
	iStateGVLData					: INT;											//State machine to handle the data on the GVL
	
	iStateModbusRead				: INT;											//State variable for Statemachine
	
	iStateModbusWrite				: INT;											//State variable for Statemachine
	
	iStateModbusError				: INT;											//State variable for Statemachine
	
	iStateModbus_CP					: INT;											//Compare State variable
	
	iMaxDcDischargeCurrentBattery	: INT;											//Variable to convert from negative to positive value
	
	diLPForGVL						: DINT;											//Loop to clean old data on GVL
	
	lrEnergyGridConsumption_CP		: LREAL;										//Energy Consumption from Grid for calculation for Workaround why Pixii send sometimes big value 
	
	lrEnergyGridProduction_CP		: LREAL;										//Energy Production from Grid for calculation for Workaround why Pixii send sometimes big value 
	int_Handshake_Counter: INT;
	i: INT;
END_VAR
VAR PERSISTENT
	diNrOfEMS_IN_CP					: DINT;											//Number of EMS what control this Device to compare with the original
END_VAR

//Creator : Stefan Lackner (based on Pixii V2.3)
//Company : EfficientIO
//Date : 02.06.2024
//Version : 1.0.0.0

//With this function its possible to read out values from the Pixii Powerbox from the factory Pixii
//Its also possible to controll the power in and out from Battery if its necessary.

//NOTE for diNr.....Designation => 
//_IN = Here Data come in from other Functions or go out to other functions about the GVL
//_OUT = Here Data go out to other functions about the GVL

(*------------------------------------------------------------------------------------------General Input Part---------------------------------------------------------------------------------------------*)

//Check limitation
diNrOfEMS_IN := LIMIT(0,diNrOfEMS_IN,Constants_Energy.diMaxNumberOfEMS);
	
(*-------------------------------------------------------------Calcualte the number of Battery system---------------------------------------------------------------*)

fbNumberDeviceBattery(
	diActualNumberOfDevices:= Lynus_Standards.GVL_Energy.stNumberOfDevices.diNumberOfBatterys, 
	diMaxNumberOfDevices:= Constants_Energy.diMaxNumberOfBatterys, 
	udiCounterOnlineChange:= TwinCAT_SystemInfoVarList._AppInfo.OnlineChangeCnt, 
	bNumberIsCalculatet=> , 
	bFPNumberIsCalculatet=> , 
	bOnlineChange=> , 
	diNumberForThisDevice=> diNrOfBatt_OUT, 
	diNumberOfTotalDevices=> );

//Write new Numer on GVL
IF fbNumberDeviceBattery.bFPNumberIsCalculatet THEN
	Lynus_Standards.GVL_Energy.stNumberOfDevices.diNumberOfBatterys := fbNumberDeviceBattery.diNumberOfTotalDevices;	
END_IF

//Delete old Number on GVL
IF fbNumberDeviceBattery.bOnlineChange THEN 
	Lynus_Standards.GVL_Energy.stNumberOfDevices.diNumberOfBatterys := diNrOfBatt_OUT;	
		iStateGVLData := 1; 
END_IF

fbNumberDeviceBatteryInvert(
	diActualNumberOfDevices:= Lynus_Standards.GVL_Energy.stNumberOfDevices.diNumberOfBatteryInverters, 
	diMaxNumberOfDevices:= Constants_Energy.diMaxNumberOfBatteryInverters, 
	udiCounterOnlineChange:= TwinCAT_SystemInfoVarList._AppInfo.OnlineChangeCnt, 
	bNumberIsCalculatet=> , 
	bFPNumberIsCalculatet=> , 
	bOnlineChange=> , 
	diNumberForThisDevice=> diNrOfBattInverter_OUT, 
	diNumberOfTotalDevices=> );

//Write new Numer on GVL
IF fbNumberDeviceBatteryInvert.bFPNumberIsCalculatet THEN
	Lynus_Standards.GVL_Energy.stNumberOfDevices.diNumberOfBatteryInverters := fbNumberDeviceBatteryInvert.diNumberOfTotalDevices;	
END_IF

//Delete old Number on GVL
IF fbNumberDeviceBatteryInvert.bOnlineChange THEN 
	Lynus_Standards.GVL_Energy.stNumberOfDevices.diNumberOfBatteryInverters := diNrOfBattInverter_OUT;	
	iStateGVLData := 1; 
END_IF

fbNumberDeviceGrid(
	diActualNumberOfDevices:= Lynus_Standards.GVL_Energy.stNumberOfDevices.diNumberOfElectricMeters, 
	diMaxNumberOfDevices:= Constants_Energy.diMaxNumberOfElectricMeters, 
	udiCounterOnlineChange:= TwinCAT_SystemInfoVarList._AppInfo.OnlineChangeCnt, 
	bNumberIsCalculatet=> , 
	bFPNumberIsCalculatet=> , 
	bOnlineChange=> , 
	diNumberForThisDevice=> diNrOfEM_OUT_Grid, 
	diNumberOfTotalDevices=> );

//Write new Numer on GVL
IF fbNumberDeviceGrid.bFPNumberIsCalculatet THEN
	Lynus_Standards.GVL_Energy.stNumberOfDevices.diNumberOfElectricMeters := fbNumberDeviceGrid.diNumberOfTotalDevices;	
END_IF			

(*-------------------------------------------------------------Service from Backend is ready and check the connection to backend for dissabel/enable Function---------------------------------------------------------------*)

//Try to reset the variable for connection on the GVL. When all is normal then the Lynus Mqtt connection function set this variable to true in the next cycle
//When we have no connection to the backend then after Lynus_Standards.Constants_General.tTimeDissableLynusFunctions days the Function is dissabled with all of his functionalities
timResetConnectionOnGVL(	IN:= NOT timResetConnectionOnGVL.Q, 
							PT:= T#1H, 
							Q=> , 
							ET=> );
IF timResetConnectionOnGVL.Q THEN 
	Lynus_Standards.GVL_Communicator.bStateConnectionToEnableFunctions := FALSE; 
END_IF
IF NOT Lynus_Standards.GVL_Communicator.bStateConnectionToEnableFunctions THEN 
	timDissableFunctions.IN := TRUE; 
ELSE 
	timDissableFunctions.IN := FALSE; 
END_IF  
timDissableFunctions(	IN:= , 
						PT:= Lynus_Standards.Constants_General.tTimeDissableLynusFunctions, 
						Q=> ,
						ET=> );
			
(*------------------------------------------------------------------------------------------State Machine Read---------------------------------------------------------------------------------------------*)

//When the function is not enabled then the fronius control by himself without modbus tcp connection
IF NOT bEnable OR timDissableFunctions.Q THEN 
	bActivateControl := FALSE; 
END_IF

// limit manual setpoint +/- 320 kW
i_SetpointPower_Manual_kW:=LIMIT(-320,i_SetpointPower_Manual_kW,320);

//Start the Statemachine
FPEnable(CLK:= bEnable, Q=> );
FPActivateControl(CLK:= bActivateControl, Q=> );
FNTimDissable(CLK:= timDissableFunctions.Q, Q=> );
IF (FPEnable.Q AND iStateModbusRead = 0 AND iStateModbusRead = 0 AND iStateModbusError = 0) OR
	(bEnable AND FPActivateControl.Q AND iStateModbusRead = 0 AND iStateModbusRead = 0 AND iStateModbusError = 0) OR
	(bEnable AND FNTimDissable.Q AND iStateModbusRead = 0 AND iStateModbusRead = 0 AND iStateModbusError = 0) THEN 
		iStateModbusRead := 1; 
END_IF
IF NOT bEnable OR NOT bActivateControl THEN 
	iStateModbusRead := 0; 
	iStateModbusWrite := 0; 
	iStateModbusError := 0; 
END_IF

//Timer for delay
timDelay(	IN:= , 
			PT:= T#500MS, 
			Q=> , 
			ET=> );

//Timer for Timeout in Statemachine
IF 	(iStateModbusRead > 0 AND iStateModbusRead <= 2 AND iStateModbusRead = iStateModbus_CP) OR
	(iStateModbusWrite > 0 AND iStateModbusWrite <= 1 AND iStateModbusWrite = iStateModbus_CP) THEN
		timTimeout.IN := TRUE;
ELSE	
		timTimeout.IN := FALSE;
END_IF 
IF iStateModbusRead = 0 AND iStateModbusWrite = 0 THEN 
	timTimeout.IN := FALSE; 
END_IF
timTimeout(	IN:= , 
			PT:= T#20S, 
			Q=> , 
			ET=> );

CASE iStateModbusRead OF
	
	0://Init State
		iStateModbus_CP := 0;
		timDelay.IN := FALSE;
			
		stDataPixii.eBatteryState := E_Pixii_BatteryState.eNoDataReceived;
		stDataPixii.eOperatingState := E_Pixii_OperatingState.eNoDataReceived;	
		stDataPixii.bFunctionIsActive := FALSE;
			
		fbMBRead_FC3.bExecute := FALSE;
		fbMBWrite_FC6.bExecute := FALSE;
		// clear buffer	
		FOR i:= 1 TO 125 BY 1 DO
			arrBuffer_FC3[i] := 0;
		END_FOR
	1://Read first data part
		stDataPixii.bFunctionIsActive := TRUE;
		iStateModbus_CP := iStateModbusRead;
		
		//Reset Write
		fbMBWrite_FC6.bExecute := FALSE;
		wordBuffer_FC6 := 0; 
		
		//Start Read
		fbMBRead_FC3.nQuantity := 80;
		fbMBRead_FC3.nMBAddr := 40121;
		fbMBRead_FC3.bExecute := TRUE;
			
		IF fbMBRead_FC3.bBusy THEN 
			timDelay.IN := TRUE; 
		END_IF
		
		//Wait for Delay, copy Data and then next step
		IF NOT fbMBRead_FC3.bBusy AND NOT fbMBRead_FC3.bError AND timDelay.Q THEN
			
		
			//Max Charge Power (in W)
			fbBatteryInverter.rMaxChargePowerBattInverter := INT_TO_REAL(WORD_TO_INT(arrBuffer_FC3[5])) * EXPT(10,INT_TO_REAL(WORD_TO_INT(arrBuffer_FC3[55]))); 
			//Max Discharge Power (in W)
			fbBatteryInverter.rMaxDischargePowerBattInverter := INT_TO_REAL(WORD_TO_INT(arrBuffer_FC3[6])) * EXPT(10,INT_TO_REAL(WORD_TO_INT(arrBuffer_FC3[55]))); 
			
			
			r_MaxChargePower_W := LIMIT (0,r_MaxChargePower_W,fbBatteryInverter.rMaxChargePowerBattInverter);
			r_MaxDischargePower_W := LIMIT (0,r_MaxDischargePower_W,fbBatteryInverter.rMaxDischargePowerBattInverter);
			
			IF m_ManualChargeDischargeMax THEN
				fbBatteryInverter.rMaxChargePowerBattInverter := r_MaxChargePower_W;
				fbBatteryInverter.rMaxDischargePowerBattInverter := r_MaxDischargePower_W;
			END_IF
				
			//SOC (No Scalefactor. Is %)	
			fbBattery.dwBatterySOC := INT_TO_DWORD(WORD_TO_INT(arrBuffer_FC3[12])) *  LREAL_TO_DWORD(EXPT(10,INT_TO_DWORD(WORD_TO_INT(arrBuffer_FC3[57]))))  ;
			fbBatteryInverter.dwBatterSOC := fbBattery.dwBatterySOC;
			//Battery State
			CASE  arrBuffer_FC3[22] OF
				0: stDataPixii.eBatteryState := E_Pixii_BatteryState.eNoDataReceived;
				1: stDataPixii.eBatteryState := E_Pixii_BatteryState.eDisconnected;
				2: stDataPixii.eBatteryState := E_Pixii_BatteryState.eInitializing;
				4: stDataPixii.eBatteryState := E_Pixii_BatteryState.eConnected;
				8: stDataPixii.eBatteryState := E_Pixii_BatteryState.eStandby;
				16: stDataPixii.eBatteryState := E_Pixii_BatteryState.eSoCProtection;
				32: stDataPixii.eBatteryState := E_Pixii_BatteryState.eSuspending;
				64: stDataPixii.eBatteryState := E_Pixii_BatteryState.eFault;			
			END_CASE

			//Battery Capacity in Wh (in Wh), but make the calculation for kWh
			lrMaxCapacityBattery_OUT := INT_TO_REAL(WORD_TO_INT(arrBuffer_FC3[4])) * EXPT(10,INT_TO_REAL(WORD_TO_INT(arrBuffer_FC3[54]))); 
			lrMaxCapacityBattery_OUT := lrMaxCapacityBattery_OUT / 1000;
			//Battery Current (in A)
			fbBattery.lrBatteryCurrent := INT_TO_REAL(WORD_TO_INT(arrBuffer_FC3[45])) * EXPT(10,INT_TO_REAL(WORD_TO_INT(arrBuffer_FC3[62]))); 
(* CHECK if PIXII NEEDS THAT			
			//Change the sign because in view from the Battery - is discharge and + is charge. But we use vice versa	
			fbBattery.lrBatteryCurrent := fbBattery.lrBatteryCurrent * - 1; 
*)			
			//Battery Voltage 
			fbBattery.rBatteryVoltage := INT_TO_REAL(WORD_TO_INT(arrBuffer_FC3[35])) * EXPT(10,INT_TO_REAL(WORD_TO_INT(arrBuffer_FC3[60]))); 
			//Max Charge Current (in A)
			fbBattery.rMaxDcChargeCurrentBattery := INT_TO_REAL(WORD_TO_INT(arrBuffer_FC3[46])) * EXPT(10,INT_TO_REAL(WORD_TO_INT(arrBuffer_FC3[63]))); 

			//Max Discharge Current (in A)
			fbBattery.rMaxDcDischargeCurrentBattery := INT_TO_REAL(WORD_TO_INT(arrBuffer_FC3[47])) * EXPT(10,INT_TO_REAL(WORD_TO_INT(arrBuffer_FC3[63]))); 
// not needed for pixii			//Its allways a negative raw value
// not needed for pixii				iMaxDcDischargeCurrentBattery := iMaxDcDischargeCurrentBattery * - 1;
//					fbBattery.rMaxDcDischargeCurrentBattery := INT_TO_REAL(iMaxDcDischargeCurrentBattery) * 100; 
					
			CASE  arrBuffer_FC3[70] OF
				0: stDataPixii.eBasicAggregatorState := E_Pixii_BasicAggregatorState.eUnkown;
				1: stDataPixii.eBasicAggregatorState := E_Pixii_BasicAggregatorState.eOff;
				2: stDataPixii.eBasicAggregatorState := E_Pixii_BasicAggregatorState.eOn;
				3: stDataPixii.eBasicAggregatorState := E_Pixii_BasicAggregatorState.eFull;
				4: stDataPixii.eBasicAggregatorState := E_Pixii_BasicAggregatorState.eFault;
	
			END_CASE

			//Go to Next Step
			fbMBRead_FC3.bExecute := FALSE;
			timDelay.IN := FALSE;		
			iStateModbusRead := 2;
		END_IF
		
//			Not needed I think
//			//Pixii Battery Error
//			IF NOT fbMBRead_FC3.bBusy AND NOT fbMBRead_FC3.bError AND timDelay.Q AND stDataPixii.eBatteryState = E_Pixii_BatteryState. THEN
//				iStateModbusError := 300;
//				stDataPixii.eErrorState := E_Pixii_Error.ePixiiError;
//			END_IF
		
		//Error or Timeout
		IF FPError_FC_3.Q OR timTimeout.Q THEN
			iStateModbusError := 300;
			stDataPixii.eErrorState := E_Pixii_Error.eModbusTCPError;
		END_IF
	
	2://Wait 1 Step to reset the delay counter befor start to write
		iStateModbus_CP := iStateModbusRead;
		// clear buffer	
		FOR i:= 1 TO 125 BY 1 DO
			arrBuffer_FC3[i] := 0;
		END_FOR		
		iStateModbusRead := 10;	
		
	10://Read second data part
		iStateModbus_CP := iStateModbusRead;
		
		//Start Read
		fbMBRead_FC3.nQuantity := 51;
		fbMBRead_FC3.nMBAddr := 40069;
		fbMBRead_FC3.bExecute := TRUE;
			
		IF fbMBRead_FC3.bBusy THEN 
			timDelay.IN := TRUE; 
		END_IF
		
		//Wait for Delay, copy Data and then next step
		IF NOT fbMBRead_FC3.bBusy AND NOT fbMBRead_FC3.bError AND timDelay.Q THEN
			
			//inverter Temperature (in °C)
			fbBattery.lrBatteryTemp := INT_TO_REAL(WORD_TO_INT(arrBuffer_FC3[34])) *  EXPT(10,INT_TO_REAL(WORD_TO_INT(arrBuffer_FC3[38])))  ;
			//Operating State
			CASE  arrBuffer_FC3[39] OF
				0:	stDataPixii.eOperatingState := E_Pixii_OperatingState.eNoDataReceived;
				1:	stDataPixii.eOperatingState := E_Pixii_OperatingState.eSleeping;
				2:	stDataPixii.eOperatingState := E_Pixii_OperatingState.eStarting;
				3:	stDataPixii.eOperatingState := E_Pixii_OperatingState.eMPPT;
				4:  stDataPixii.eOperatingState := E_Pixii_OperatingState.eThrottled;
				5: stDataPixii.eOperatingState := E_Pixii_OperatingState.eShuttingDown;
				6: stDataPixii.eOperatingState := E_Pixii_OperatingState.eFault;
				7: stDataPixii.eOperatingState := E_Pixii_OperatingState.eStandby;
			END_CASE
(*					eNoDataReceived := 0,
					eSleeping := 1,
					eStarting := 2,
					eMPPT := 3,
					eThrottled := 4,
					eShuttingDown := 5,
					eFault := 6,
					eStandby := 7 *)

			fbEMPower.lrCurrentL1 := INT_TO_REAL(WORD_TO_INT(arrBuffer_FC3[4])) *  EXPT(10,INT_TO_REAL(WORD_TO_INT(arrBuffer_FC3[7])))  ;
			fbEMPower.lrCurrentL2 := INT_TO_REAL(WORD_TO_INT(arrBuffer_FC3[5])) *  EXPT(10,INT_TO_REAL(WORD_TO_INT(arrBuffer_FC3[7])))  ;
			fbEMPower.lrCurrentL3 := INT_TO_REAL(WORD_TO_INT(arrBuffer_FC3[6])) *  EXPT(10,INT_TO_REAL(WORD_TO_INT(arrBuffer_FC3[7])))  ;
			fbEMPower.lrVoltageL1N := INT_TO_REAL(WORD_TO_INT(arrBuffer_FC3[11])) *  EXPT(10,INT_TO_REAL(WORD_TO_INT(arrBuffer_FC3[14])))  ;
			fbEMPower.lrVoltageL2N := INT_TO_REAL(WORD_TO_INT(arrBuffer_FC3[12])) *  EXPT(10,INT_TO_REAL(WORD_TO_INT(arrBuffer_FC3[14])))  ;
			fbEMPower.lrVoltageL3N := INT_TO_REAL(WORD_TO_INT(arrBuffer_FC3[13])) *  EXPT(10,INT_TO_REAL(WORD_TO_INT(arrBuffer_FC3[14])))  ;
			fbEMPower.lrVoltageL1L2 := fbEMPower.lrVoltageL1N * 1.73;
			fbEMPower.lrVoltageL2L3 := fbEMPower.lrVoltageL2N * 1.73;
			fbEMPower.lrVoltageL3L1 := fbEMPower.lrVoltageL3N * 1.73;
			fbEMPower.lrPowerTotal	:= INT_TO_REAL(WORD_TO_INT(arrBuffer_FC3[15])) *  EXPT(10,INT_TO_REAL(WORD_TO_INT(arrBuffer_FC3[16])))  ;
			fbEMPower.lrFrequency	:= INT_TO_REAL(WORD_TO_INT(arrBuffer_FC3[17])) *  EXPT(10,INT_TO_REAL(WORD_TO_INT(arrBuffer_FC3[18])))  ;
			fbEMPower.lrApparentPowerTotal := INT_TO_REAL(WORD_TO_INT(arrBuffer_FC3[19])) *  EXPT(10,INT_TO_REAL(WORD_TO_INT(arrBuffer_FC3[20])))  ;
			fbEMPower.lrReactivePowerTotal := INT_TO_REAL(WORD_TO_INT(arrBuffer_FC3[21])) *  EXPT(10,INT_TO_REAL(WORD_TO_INT(arrBuffer_FC3[22])))  ;
			
			
			
			//Go to Next Step
			fbMBRead_FC3.bExecute := FALSE;
			timDelay.IN := FALSE;		
			iStateModbusRead := 11;
		END_IF
		
		//Error or Timeout
		IF FPError_FC_3.Q OR timTimeout.Q THEN
			iStateModbusError := 300;
			stDataPixii.eErrorState := E_Pixii_Error.eModbusTCPError;
		END_IF
	
	11://Wait 1 Step to reset the delay counter befor start to write
		iStateModbus_CP := iStateModbusRead;
	
		iStateModbusWrite := 1;
		iStateModbusRead := - 1;	
					
END_CASE

(*----------------------------------------------------------------------------------------Battery Inverter Function----------------------------------------------------------------------------------------------*)

//Error and Reset
timErrorMTCP(	IN:= stDataPixii.bError AND stDataPixii.eErrorState = E_Pixii_Error.eModbusTCPError, 
				PT:= T#5S, 
				Q=> , 
				ET=> );

IF timDissableFunctions.Q THEN 
	fbBatteryInverter.bWarning := TRUE; 
	fbBatteryInverter.iWarningCode := 0; 
ELSE 
	fbBatteryInverter.bWarning := FALSE; 
END_IF 
IF (stDataPixii.bError  OR timErrorMTCP.Q OR Lynus_Standards.GVL_Energy.stNumberOfDevices.diNumberOfBatteryInverters > Constants_Energy.diMaxNumberOfBatteryInverters) THEN 
	fbBatteryInverter.bError := TRUE; 
ELSE 
	fbBatteryInverter.bError := FALSE; 
END_IF	
IF Lynus_Standards.GVL_Energy.stNumberOfDevices.diNumberOfBatteryInverters > Constants_Energy.diMaxNumberOfBatteryInverters THEN 
	fbBatteryInverter.iErrorCode := 1;
ELSIF stDataPixii.bError THEN 
	fbBatteryInverter.iErrorCode := 0; 
END_IF  

//Autoreset after Error, because Pixii deleiver somtimes a Error and they dont know why.....
timReset(	IN:= stDataBattInverter.byErrorWarning <> 0 AND NOT timReset.Q, 
			PT:= T#1S, 
			Q=> , 
			ET=> );	
		
//Island mode active  ---> no island mode for pixii
fbBatteryInverter.bWorkOnIslandMode := FALSE; 

		
//Function
fbBatteryInverter(
	bEnable:= bEnable AND NOT timDissableFunctions.Q, 
	bInverterOnOff:= TRUE, 
	bError:= , 
	bWarning:= , 
	bReset:= bReset OR timReset.Q,  
	bWorkOnIslandMode:= , 
	bWriteWithDelay:= TRUE, 
	byPriority:= byPriority, 
	byReserveSOCEPO:= Lynus_Standards.GVL_Energy.stDataOfBatteryInverters[diNrOfEMS_IN,diNrOfBattInverter_OUT].byReserveSOCEPO, 
	byMaxDepthOfDischargeEPO:= Lynus_Standards.GVL_Energy.stDataOfBatteryInverters[diNrOfEMS_IN,diNrOfBattInverter_OUT].byMaxDepthOfDischargeEPO, 
	iErrorCode:= , 
	iWarningCode:= , 
	dwBatterSOC:= , 
	rTargetPower:= Lynus_Standards.GVL_Energy.stDataOfBatteryInverters[diNrOfEMS_IN,diNrOfBattInverter_OUT].rTargetPowerEMS, 
	lrActualBatteryPower:= fbBattery.lrBatteryCurrent * fbBattery.rBatteryVoltage, 
	rMaxChargePowerBattInverter:= , 
	rMaxDischargePowerBattInverter:= , 
	lrBattInverterPowerOnIslandMode:= 0, 
	lrBattInverterPowerOnNormalMode:= 0, 
	tTimDelayOutput:= T#5S, 
	stDataBattInvertOut=> , 
	stDataBattInvertOutDelay=> stDataBattInverter);

//Controller to hold the Battery Current to 0 and take the rest from the Grid. (Avoid discharge in standby or when reaching the reserve charge for EPO)
timSetStandbyCntrl(	IN:= fbBatteryInverter.stDataBattInvertOut.rTargetPower = 0, 
					PT:= T#5S, 
					Q=> , 
					ET=> );

IF timSetStandbyCntrl.Q AND bEnable AND bActivateControl THEN
	fbPIDChrgStandby.bEnable := TRUE;
	//Charge the Battery when its under the reserve for SOC
	IF fbBatteryInverter.dwBatterSOC < fbBatteryInverter.byReserveSOCEPO THEN
		fbPIDChrgStandby.rSetpoint := (fbBattery.stDataBatteryOut.rMaxDcChargeCurrent * 0.1) * - 1; 	
	ELSE
		fbPIDChrgStandby.rSetpoint := 0;	
	END_IF		 
ELSE
	fbPIDChrgStandby.bEnable := FALSE;
END_IF

fbPIDChrgStandby( 
	bEnable:= , 
	rSetpoint:= , 
	udiIValue:= 750, 
	udiDValue:= 0, 
	udiDamping:= 0, 
	rPValue:= 0.32, 
	rMaxValue:= 0, 
	rMinValue:= ((fbBatteryInverter.rMaxChargePowerBattInverter / 100) * - 1) / 2, 
	rNeutralZone:= 0.1, 
	bDirection:= FALSE, 
	rActualValue:= LREAL_TO_REAL(fbBattery.stDataBatteryOut.lrCurrent), 
	rQController=> );	

//Set the Target power to a fixed value when the controller is acitve
IF fbPIDChrgStandby.bEnable THEN 
	stDataBattInverter.rTargetPower := - 1;
END_IF
	
(*----------------------------------------------------------------------------------------Battery Function----------------------------------------------------------------------------------------------*)

